(* PLC project LorochCxPlc_1, Beckhoff Automation GmbH TwinCAT PLC Control 3.5.13.20 *)
(* stored: creationDateTime 2021-05-25T13:03:07.2332886, modificationDateTime 2021-05-25T13:03:07.2402695 *)

FUNCTION_BLOCK FB_SFC_CHIPBREAKER_AUTO
(*---------------------------------------------------------------------------------------------------------------------------------------------------------------------------

			Date	I	version	I	remarks
					I			I
					I			I
					I			I
----------------------------------------------------------------------------------------------------------------------------------------------------------------------------*)
VAR_INPUT
				(*Positionierung Manuelle*)
				YDistanceToTouchPos					:	LREAL;
				ManPosActive							:	BOOL;
				XMoveManual							:	BOOL;
				SimpleTouch								:	BOOL;			(*Only 1 Touch*)
				KeyNextStep								:	BOOL;
				YrefPos									:	LREAL;			(*Reference Position  of Y-Axis)*)
				DoubleTouch								:	 BOOL;
				WorkingAngle							:	LREAL;
				Reset									:	 BOOL;
				PauseSwitchActive						:	 BOOL;
				MachineStateSafetyStateActive				:	 BOOL;
				MachineStateSharpenerDoorIsClosed		:        	BOOL;
				Start										:	 BOOL;
				AutomaticMode							:	 BOOL;
				ActualSawBlade							:	ST_SawBlade;
				ActualGrindingWheel						:	ST_GrindingWheel;
				ActualJob								:	ST_Job;
				AStartPos								:	 LREAL;				(*Rear Pos*)
				ChamferSideString						:	 STRING;
				ToothPitch								:	 LREAL;
				GrindingDirCW							:	 BOOL;
				DeltaMax								:	LREAL;
				TeethNumber								:	 INT;
				Stepper									:	 BOOL;							(*Using Servo Motor*)
				CbaPneumatic							:	BOOL;
				Zx										:	LREAL;							(*Z_Axis Corrector*)
				(*stepper-servo*)
				MarginRearValue							:	LREAL;							(*this value: Randabstand rear side to be set by the user*)
				MarginFrontValue							:	LREAL;							(*this value: Randabstand front side to be set by the user*)
				CbaMotionType							:	E_MotionType;
END_VAR
VAR_OUTPUT
				ActualStep								:	 INT;
				ErrorID									:	 DINT;
				ErrorOut									:	 BOOL;
				Paused									: 	BOOL;
				PauseRequest							:	 BOOL;
				PauseAvailable							:	 BOOL;
				CammingActive							:	 BOOL;
				ActualRevolutions							:     	UINT;
				ZStartposBuffered							:	 LREAL;
				ActualInfeed								:	LREAL;							(* actual infeed *)
				PartialInfeed								:	LREAL;
				ToothCount								:	INT;
				ZaxisCbaLimit							:	BOOL;
				CBAutoNotPossibleWithTooLargeSbDiameter	:	BOOL;
				WarningAaxisIsSlow						:	BOOL;
				CbaSpindleLowSpeedOutput				:	BOOL;

END_VAR

VAR_IN_OUT
				Done									:	BOOL;
				TouchPositionZAxis						:	LREAL;
				ChipBreakerAutoVeloTemp					:	LREAL;
				ChipBreakerManVeloOverrideFactor			:	LREAL;
END_VAR

VAR
				(*Manual Positionning*)
				RTrigConfirmTouchposZ					:	 R_TRIG;
				RTrigConfirmTouchposX					:	 R_TRIG;
				TON_Wait								:	 TON;
				DeltaXChamfering							:	 LREAL;
				ActualTeeth								:	 INT;
				SfcChipBreakerAuto						:	 FB_SUBFUNC_SEQ_CONTROL;	(* FB sfc *)
				XAxisStartPosition 							:	 LREAL;
				ZAxisStartPosition							:	 LREAL;
				ChipBreakerRear							:	 BOOL;
				StepNew									:	 INT;
				StepAction								:	 BOOL;
				StepActionImPulse						:	 BOOL;
				PauseStep								:	 INT;
				WorkingStepNo							:	 INT;
				AxisState								:	 E_StateMachineAxis;				(* check state of axis *)
				SBCircumference							:	 LREAL;
				ChipBreakerXAxisVelo						:	 LREAL;
				ChipBreakerAutoXAxisMaxVelo				: 	 LREAL;
				YAxisStartPosition							:	 LREAL;
				DegPerTeeth								:	 LREAL;
				XAxisTouchposRadio						:	 LREAL;
				TouchCorrection							:	 LREAL;
				FBCalcXOffset							:	 LREAL;
				XOffset									:	 LREAL;
				ZOffset									:	 LREAL;
				VarioCtr									:	 INT;
				VarioCtrEnd								:	 INT;
				XAxisEndPos								:	 LREAL;
				ZTouchPos								:	 LREAL;
				NumberTouch							:	 INT ;
				Delta									:         LREAL;			(*ABS(TP1-TP2)*)
				NominalTeeth							:	 LREAL;
				PauseRequested							:	 BOOL;
				PartialInfeedChangedDownfeed				:	 BOOL;
				ZAxisPausePos							:	 LREAL;
				InfeedZAxisMM							:	 LREAL;
				TouchPositionsZPlausi						:	 ARRAY[0..2] OF LREAL;
				TouchPositionsPlausibilityOK				:	 BOOL;
				TouchPositionsPlausibilityError				:	 BOOL;
				ChipBreakerFront							:	 BOOL;
				XaxisEndPOsFront						:	 LREAL;			(*X-Axis End Position After The Sharpening *)
				DeltaX									:	 LREAL;
				DeltaZ									:	 LREAL;
				YendPos								:	 LREAL;			(*End Position Y-Axis after Grinding*)
				ZAxisUpfeedMM							:	 LREAL;
				ZAxisUpfeedPosition						:	 LREAL;
				WorkingAngleRAD						:	 LREAL;
				RSS									:	 LREAL;
				BSS										:	 LREAL	;
				ChipBreakerFr							:	 BOOL	:=	TRUE;
				ChipBreakerRe							:	 BOOL	:=	FALSE ;
				NumberRevolution						:	 INT:=0	     ;
				ActualGrindingWheelThickness				:	 LREAL;
				(*Enumeration added*)
				RTrigNextStep							:	R_TRIG;
				ContinousMode							:	 BOOL;
				NextStepPulse							:	BOOL;
				XPosition								:	LREAL;
				ZPosition								:	LREAL;
				TON_Rear								:	TON;							(*Delay before the start of the Rear Side*)
				TONWaitSafetyStatePause					:	TON;
				FTRIG_STOP							:	F_TRIG;
				DeltaX_DEG								:	LREAL;
				XoffsetInGrad								:	LREAL;
				TonWaitClamping							:	TON;
				Test										:	BOOL;
				StopChipBreaker							:	BOOL;
				StartButton								:	R_TRIG;
				Stop_Manual_Pos							:	F_TRIG;
				DSSDiff									:	LREAL;
				ZPosAfterSharpening						:	LREAL;
				(*Software Limit S*)
				ZAxisLimitPos							:	BOOL;
				R_TRIG_ZlimitPos							:	R_TRIG;
				CbaLimit									:	BOOL;
				WaitAfterPause							:	TON;
				(*Vario*)
				VarioToothPitch							:	ARRAY[0..11] OF LREAL;
				VarioCtrFront1							:	INT;
				VarioCtrFront2							:	INT;
				VarioCtrRear1							:	INT;
				VarioCtrRear2							:	INT;
				GearPlayXAxis							:	LREAL;
				DifferenceMaxMinCBAGWDiameter			:	LREAL;
				(*Display Warning*)
				UIEventCBAProtection						:	FB_SUBFUNC_MESSAGE;
				ChipBreakerAutoGWwidth					:	LREAL;
				AaxisReferenceValue						:	LREAL;    (*the initial distance in MM when the axis is in home position*)
				AFront80									:	LREAL;	(*80% of the A-Axis front destination*)
				ARear80									:	LREAL;	(*80 % of the A -Axis Rear position *)
				AaxisRef80								:	LREAL;	(**)
				ARearPos								:	LREAL;
				AFrontPos								:	 LREAL;
				TonMonitoringAaxis						:	TON;
				StartMonitoringAaxis						:	BOOL;
				WarningAaxis								:	BOOL;
				RtrigAaxisIsTooSlow						:	R_TRIG;
				RtrigSpindleLowSpeedError				:	R_TRIG;
				CbaSpindleLowSpeed						:	BOOL;
				TriesNumber								:	INT;  (*Number of tries to find out the Reference position of A-axis*)
				AaxisRefPosTemp						:	LREAL;
				AaxisActPosition							:	LREAL;
				StartMovingStepByStepRear				:	BOOL; (**)
				StartMovingStepByStepFront				:	BOOL;
				ZTouchPosFirstTouchPos					:	LREAL;
				AaxisStepPositionIsReached				:	BOOL;
				WaitForAaxis								:	TON;
				StartWaitAaxis							:	BOOL;
				ZaxisFirstTouchPos						:	LREAL;
				ZNoTouch								:	LREAL;
				LastZPos								:	LREAL;
				LimitZaxis								:	LREAL;
				Zcomp									:	LREAL;
				StepperResults							:	FB_StepperResults;
				FileNameExtension						:	T_MaxString;
				StartWriting								:	BOOL;
				FileName								:	STRING;
				stTimeStruct								: 	TIMESTRUCT;
				stTimeStartM								: 	TIMESTRUCT;
				stTimeEndM								: 	TIMESTRUCT;
				ZposForCsv								:	LREAL;
				DurationAaxisMotion						:	TIME;
				StartTimeCounting							:	BOOL;
				TonCounting								:	TP;
				fbGetTime								: 	NT_GetTime;
				FirstEdgePos								:	LREAL;
				TestZ									:	BOOL;
				SecondEdge								:	LREAL;
				StepMotorNeededTimeToMove				:	TIME;
				StepMotorDestination						:	LREAL;
				AaxisTolerenceFast						:	LREAL;
				AaxisTolerenceSlow						:	LREAL;
				RTrigMonitoringCrash						:	R_TRIG;
				MonitoringTouchBack						:	LREAL;
				MonitoringTouchFront						:	LREAL;
				OperatingDirection						:	ST_OperatingDirection;
				TestCW									:	BOOL;
				TestCCW								:	BOOL;
				CalculatedXPosition,DiffXactposXcalcPos		:	LREAL;
				NumberOfTeethToAddReal					:	LREAL;
				NumberOfTeethToAdd						:	INT;
				rValueToAdd								:	LREAL;
				NombreOfRevolution						:	INT;
				GearPlayXAxisSharpChamfer				:	LREAL;
				(* Compensation *)
				NoOfActTeethCompensation				:	INT;
				XAxisNextPosition							:	LREAL;
				TestArray								:	ARRAY[0..5] OF BOOL;
END_VAR

            
	(* ---------------------------------------------------------------------------- SFC CHIPBREAKER AUTO -------------------------------------------------------------------------- *)

	(* call sfc functionblock *)
	SfcChipBreakerAuto(
						StepNew			:=	StepNew ,
						Reset			:=	Reset ,
						Step			=>	ActualStep ,
						StepAction		=>	StepAction ,
						StepActionImPulse=>	StepActionImPulse			 );


	TestZ			:=	TRUE;

	ContinousMode      := 	TRUE; 	   ;	(*TRUE; ;*)


	(*Reset the Sfc Variables*)
	IF	Reset
		THEN
			CbaSpindleLowSpeed														:=	FALSE;
			CbaSpindleLowSpeedOutput												:=	FALSE;
			StepNew																	:= 	0;
			Done																	:=	FALSE;
			ErrorOut																	:=	FALSE;
			ErrorID																	:=	0;
			StopChipBreaker															:=	FALSE;
			ZaxisCbaLimit															:=	FALSE;
			CBAutoNotPossibleWithTooLargeSbDiameter									:=	FALSE;
			MachineCtrl.Peripheral.ChipBreaker.Auto.DustFan.CmdOn						:=	FALSE;
			MachineCtrl.Peripheral.ChipBreaker.Auto.LowSpeedMonitoring.IsDeactivated		:=	FALSE;
			WarningAaxis																:=	FALSE;
			WarningAaxisIsSlow														:=	FALSE;
			MachineCtrl.ProcessControl.Warning.No										:=	0;
			StartTimeCounting															:=	FALSE;
			RTrigMonitoringCrash(CLK:=FALSE);
			MachineCtrl.State.ChipBreaker.Auto.GrindingWheelIsReady						:=	FALSE;
	END_IF;

			ChipBreakerAutoGWwidth			:=		UI.MachineSpecification.PeripheralOptional.ChipBreaker.GrindingWheel.Width.Nominal;

			AaxisTolerenceSlow				:=		0.01;
			AaxisTolerenceFast				:=		0.03;

			(*Edge distance  from ui*)


			MarginRearValue					:= 	UI.Order.Job[UI.State.ActualValues.ActualJobNumber.Maximal -1].EdgeDistance.EdgeDistanceRear;
			MarginFrontValue					:= 	UI.Order.Job[UI.State.ActualValues.ActualJobNumber.Maximal -1].EdgeDistance.EdgeDistanceFront;;


	(*###############################################A-Stepper Monitoring###############################################*)
			IF	(AxisCtrl[AxisNo.AAxis].Command.NominalValue.VeloJog <> 0)
				THEN
					IF	(StepNew <> 5030) AND
						(StepNew <> 5090)AND
						(StepNew <> 5100)
						THEN
							StepMotorNeededTimeToMove		:=
																		LREAL_TO_TIME(( ABS( AaxisActPosition -
																						StepMotorDestination ) /
																						AxisCtrl[AxisNo.AAxis].Command.NominalValue.VeloJog) );
																	;
						ELSE
							StepMotorNeededTimeToMove		:=	TIME#0.1s;
					END_IF;
				ELSE
					StepMotorNeededTimeToMove		:=	TIME#0.1s;
			END_IF;

			TonMonitoringAaxis(IN:= StartMonitoringAaxis , PT:= (StepMotorNeededTimeToMove*1000)+TIME#4s , Q=> , ET=> );


			RtrigAaxisIsTooSlow(CLK	:=	TonMonitoringAaxis.Q  , Q=> );

	(*Generate an error if the A-Axis is slow or not moving*)

	IF	RtrigAaxisIsTooSlow.Q
		THEN
			StepNew					:=	31000;
			TonMonitoringAaxis(  IN	:=	FALSE);
			RtrigAaxisIsTooSlow(CLK	:=	FALSE);
			StartMonitoringAaxis		:=	FALSE;
			WarningAaxis				:=	TRUE;
	END_IF;

	(*############################################A-Stepper Monitoring End##############################################*)

			StartButton(CLK:= MachineCtrl.Peripheral.ExternalControl.StartSwitch , Q=> );

		(*Manual Positionning*)

			ManPosActive	:=	MachineCtrl.Peripheral.ChipBreaker.Auto.PositionningMode.ManualPositionningIsActive;


		(*---------Software Limit--------------*)

			R_TRIG_ZlimitPos	(CLK :=	ZAxisLimitPos , Q=> );


		(*Controlling Z-Axis Limit Position*)
		IF	R_TRIG_ZlimitPos.Q
			THEN
				StepNew		:=	31000;
				CbaLimit		:=	TRUE;
		END_IF;

		(*Stop Button *)

		Stop_Manual_Pos(CLK:=	 (NOT PauseSwitchActive) , Q=> );

		FTRIG_STOP(CLK	:=	 (NOT PauseSwitchActive) ,
								   Q		=>		 );

		(*Z-Axis Confirm Touch Pos*)
		RTrigConfirmTouchposZ(CLK	:=	MachineCtrl.Peripheral.ExternalControl.ConfirmTouchpos	 , Q=> );

		(*X-Axis Confirm Touch Pos*)
		RTrigConfirmTouchposX(CLK	:= 	MachineCtrl.Peripheral.ExternalControl.ConfirmTouchpos, 	Q=> );


		IF	(StepNew	= 9815)
			THEN
				StartTimeCounting		:=	TRUE;
		END_IF;


	TonCounting(IN:= StartTimeCounting , PT:=TIME#180s , Q=> , ET=> );

		IF	(StepNew	= 985)
			THEN
				StartTimeCounting		:=	FALSE;
				DurationAaxisMotion	:=	TonCounting.ET;
		END_IF;


		(* r_trig next step *)
		RTrigNextStep( CLK := KeyNextStep );
		(* no confirm *)
		(*ContinousMode := FALSE;*)

;
	(*------------------------------------------Pause Requeted---------------------------------------*)

IF	(SfcChipBreakerAuto.Step	<=	1350) AND
	(SfcChipBreakerAuto.Step	>=	1300) AND
		(* pause switch is pressed *)
	(NOT PauseSwitchActive)
		THEN
			PauseRequested		:=	TRUE;
	END_IF;


IF	(SfcChipBreakerAuto.Step	= 9815)
	THEN
		IF	FTRIG_STOP.Q
		THEN
			StepNew		:=	31000;				(*Stop Routine *)
	END_IF;
END_IF;


IF	((SfcChipBreakerAuto.Step	>	1350) OR
	(SfcChipBreakerAuto.Step	<	1300))  AND(*OR*)
	( (SfcChipBreakerAuto.Step	<	90) OR
	(SfcChipBreakerAuto.Step	>	170))
	THEN
		IF	FTRIG_STOP.Q
			THEN
				StepNew		:=	31000;				(*Stop Routine *)
		END_IF;
END_IF;


IF	(SfcChipBreakerAuto.Step >=90)  AND
	(SfcChipBreakerAuto.Step <=170) AND
	Stop_Manual_Pos.Q
	THEN

				StepNew		:=	31600;				(*Direct Stop*)
END_IF;

	(*---------------------------------------ERROR------------------------------------------*)
	(*Error*)
	IF	(ChipBreakerFr AND
		ChipBreakerRe) OR
		( CbaPneumatic AND
		 Stepper)
		THEN
			StepNew		:=	25000;		(*Error*)
	END_IF;

	(* --------------------------------------sfc Reset----------------------------------------- *)

	IF	Reset
		THEN
			StepNew																	:= 	0;
			Done																	:=	FALSE;
			ErrorOut																	:=	FALSE;
			ErrorID																	:=	0;
			StopChipBreaker															:=	FALSE;
			ZaxisCbaLimit															:=	FALSE;
			CBAutoNotPossibleWithTooLargeSbDiameter									:=	FALSE;
			MachineCtrl.Peripheral.ChipBreaker.Auto.DustFan.CmdOn						:=	FALSE;
			MachineCtrl.Peripheral.ChipBreaker.Auto.LowSpeedMonitoring.IsDeactivated		:=	FALSE;
			WarningAaxis																:=	FALSE;
			AaxisStepPositionIsReached												:=	FALSE;
			StartWaitAaxis															:=	FALSE;
			ZNoTouch																:=	0;
			 MachineCtrl.Peripheral.ChipBreaker.Auto.LowSpeedMonitoring.ErrorOccured 		:=	FALSE;
			RTrigMonitoringCrash(CLK:=FALSE);
			MachineCtrl.State.ChipBreaker.Auto.GrindingWheelIsReady						:=	FALSE;
	END_IF;






	(*Test low speed warning and instead error*)

	RtrigSpindleLowSpeedError(CLK:= MachineCtrl.Peripheral.ChipBreaker.Auto.LowSpeedMonitoring.ErrorOccured , Q=> );

	IF	RtrigSpindleLowSpeedError.Q
		THEN
			 StepNew			:=	31000;
			CbaSpindleLowSpeed	:=	 TRUE;
	END_IF;



	ZAxisLimitPos		:=	(Axis[AxisNo.ZAxis].NcToPlc.ActPos <=  (UI.Order.SawBladeHolder.SawBladeLimitation[SBHChipBreakerAutoProtectionIndex].SawBladeDiameter.Minimal)) AND
							(StepNew >=85);

	(*---------------------------------------- pause------------------------------------------- *)

	IF	(SfcChipBreakerAuto.Step	<=	1350) AND
		(SfcChipBreakerAuto.Step	>=	1300)
		THEN
		IF	PauseAvailable AND
			(* pause switch is pressed *)
			(NOT PauseSwitchActive)
			THEN
				PauseRequested			:=	TRUE;
		END_IF;
	END_IF;



	CASE	SfcChipBreakerAuto.Step	OF

		(*------------------------------------------------------------------------ init Step - Reset all------------------------------------------------------------------------  *)
	0	:		(* action: predefine values *)
					CBAutoNotPossibleWithTooLargeSbDiameter							:=	FALSE;
					IF	StepActionImPulse
						THEN
							(* set axis state for check *)
								AxisState	:=	STATE_DISABLED;

							(* Reset x-axis *)
								AxisCtrl[AxisNo.XAxis].Command.OperationMode.CmdPowerOn				:=	FALSE;
								AxisCtrl[AxisNo.XAxis].Command.OperationMode.CmdMoveAbsolut			:=	FALSE;
								AxisCtrl[AxisNo.XAxis].Command.OperationMode.CmdCamming				:=	FALSE;

							(* Reset Z-axis *)
								AxisCtrl[AxisNo.ZAxis].Command.OperationMode.CmdPowerOn				:=	FALSE;
								AxisCtrl[AxisNo.ZAxis].Command.OperationMode.CmdMoveAbsolut			:=	FALSE;
								AxisCtrl[AxisNo.ZAxis].Command.OperationMode.CmdCamming				:=	FALSE;
							(*Reset A-Axis*)
								AxisCtrl[AxisNo.AAxis].Command.OperationMode.CmdPowerOn				:=	FALSE;
								AxisCtrl[AxisNo.AAxis].Command.OperationMode.CmdMoveAbsolut			:=	FALSE;
								AxisCtrl[AxisNo.AAxis].Command.OperationMode.CmdCamming				:=	FALSE;
								AxisCtrl[AxisNo.AAxis].Command.OperationMode.CmdJog					:=	FALSE;

								MachineCtrl.Peripheral.ChipBreaker.Auto.DustFan.CmdOn					:=	FALSE;
								CBAutoNotPossibleWithTooLargeSbDiameter								:=	FALSE;
								MachineCtrl.State.ChipBreaker.Auto.PauseIsActive							:=	FALSE;
								MachineCtrl.Peripheral.ExternalControl.StatusLedOnTouch1					:=	FALSE;
								MachineCtrl.Peripheral.ExternalControl.StatusLedOnTouch2					:=	FALSE;

								MachineCtrl.Peripheral.ChipBreaker.Auto.LowSpeedMonitoring.IsDeactivated	:=	FALSE;
								 MachineCtrl.Peripheral.ChipBreaker.Auto.LowSpeedMonitoring.ErrorOccured 	:=	FALSE;

								Done						:=	FALSE;
								ErrorOut						:=	FALSE;
								ErrorID						:=	0;
								ActualTeeth					:=	0;
								Paused						:=	FALSE;
								PauseStep					:=	0;
								PauseAvailable				:=	FALSE;
								PauseRequest				:=	FALSE;
								PauseRequested				:=	FALSE;
								WorkingStepNo				:=	1;
								CammingActive				:=	FALSE;
								NumberTouch				:=	0;
								Delta						:=	0;
								NumberRevolution			:=	0;
								SimpleTouch					:=	FALSE;				(*OnlyOne Touch*)
								DoubleTouch					:=	FALSE;				(*We Requie 2 Touchs*)
								ErrorOut						:=	FALSE;
								NumberTouch				:=	0;
								ActualRevolutions				:=	0;
								StopChipBreaker				:=	FALSE;
								KeyNextStep					:=	FALSE;
								(*Positionning Type*)
								ManPosActive				:=	FALSE;
								(* status led touching *)
								CbaSpindleLowSpeed			:=	FALSE;
								CbaSpindleLowSpeedOutput	:=	FALSE;
								StopChipBreaker				:=	FALSE;
								CbaLimit						:=	FALSE;
								ZaxisCbaLimit				:=	FALSE;
								WarningAaxis					:=	FALSE;
								WarningAaxisIsSlow			:=	FALSE;
								StartMonitoringAaxis			:=	FALSE;
								StartMovingStepByStepRear	:=	FALSE;
								StartMovingStepByStepFront	:=	FALSE;
								TriesNumber					:=	0;
								AaxisStepPositionIsReached	:=	FALSE;
								StartWaitAaxis				:=	FALSE;
								ZNoTouch					:=	0;
								ZposForCsv					:=	0;
								StartWriting					:=	FALSE;
								RTrigMonitoringCrash(CLK:=FALSE);
								TestCW						:=	FALSE;
								TestCCW					:=	FALSE;
					END_IF;

					(* transition *)
					IF	StepAction AND
						(NOT StepActionImPulse) AND
						(* stop switch not pressed *)
							PauseSwitchActive
						THEN
							StepNew	:= 10;									(* -> wait for Start *)
					END_IF;
		(*-------------------------------------------------------------  wait for Start----------------------------------------------------------------- *)
	10	:
					(* transition:  *)
					IF	StepAction AND
						(NOT StepActionImPulse) AND
						(* recut/resharp only in automatic mode *)
							AutomaticMode AND
						(* Start sfc from external *)
							Start AND
						(* machine door is closed *)
							MachineStateSharpenerDoorIsClosed AND
						(* safe state are disabled *)
							(NOT MachineStateSafetyStateActive) AND
						 (* stop switch not pressed *)
							(PauseSwitchActive)
						THEN
							StepNew									:= 	20;									(* -> Enable X-axis ,Z-axis and A -Axis*)
							ChipBreakerFr							:=	TRUE;
							ChipBreakerRe							:=	FALSE;
							StopChipBreaker							:=	FALSE;
							KeyNextStep								:=	FALSE;
							ErrorOut									:=	FALSE;
							ZaxisCbaLimit							:=	FALSE;
							CBAutoNotPossibleWithTooLargeSbDiameter	:=	FALSE;
							AaxisRefPosTemp						:=	UI.MachineSpecification.PeripheralOptional.ChipBreaker.Notch.SBEdgeOffset;			(*Reference Value of the A-Axis*)
							AaxisReferenceValue						:=	AaxisRefPosTemp;
							AaxisStepPositionIsReached				:=	FALSE;
							StartWaitAaxis							:=	FALSE;
							ZNoTouch								:=	0;
							StartWriting								:=	FALSE;
							 MachineCtrl.Peripheral.ChipBreaker.Auto.LowSpeedMonitoring.ErrorOccured 	:=	FALSE;
							MachineCtrl.State.ChipBreaker.Auto.GrindingWheelIsReady					:=	FALSE;
					END_IF;

		(*------------------------------------------------------------Wait For User Interaction--------------------------------------------------------------*)
	20:			IF	StepActionImpulse
					THEN
						NextStepPulse		:=	TRUE;
					END_IF;

				IF	StepAction AND
					( RTrigNextStep.Q OR
					ContinousMode )
					THEN
						StepNew				:= 	22;
						NextStepPulse		:=	FALSE;
						ErrorOut				:=	FALSE;
				END_IF;

		(*---------------------------------------------------------------- action: Enable x +z+a Axis-----------------------------------------------------------*)
	22	:		(*Action*)
					ErrorOut					:=	FALSE;
					IF	StepActionImPulse
						THEN
							(* set axis state for check *)
								AxisState	:=	STATE_WAIT_NEWOPERATION;
							(* x-axis - Enable *)
								AxisCtrl[AxisNo.XAxis].Command.OperationMode.CmdPowerOn			:=	TRUE;
								AxisCtrl[AxisNo.XAxis].Command.OperationMode.CmdMoveAbsolut		:=	FALSE;
								AxisCtrl[AxisNo.XAxis].Command.OperationMode.CmdCamming			:=	FALSE;
								AxisCtrl[AxisNo.XAxis].Command.ExternalControl.override				:=	100;
							(* Z-axis - Enable *)
								AxisCtrl[AxisNo.ZAxis].Command.OperationMode.CmdPowerOn			:=	TRUE;
								AxisCtrl[AxisNo.ZAxis].Command.OperationMode.CmdMoveAbsolut		:=	FALSE;
								AxisCtrl[AxisNo.ZAxis].Command.OperationMode.CmdCamming			:=	FALSE;
								AxisCtrl[AxisNo.ZAxis].Command.ExternalControl.override				:=	100;
							(* Axis Is Used--> Axis Enable*)
								IF	Stepper
									THEN
							(*A-Axis- Enable*)
								AxisCtrl[AxisNo.AAxis].Command.OperationMode.CmdPowerOn			:=	TRUE;
								AxisCtrl[AxisNo.AAxis].Command.OperationMode.CmdMoveAbsolut		:=	FALSE;
								AxisCtrl[AxisNo.AAxis].Command.OperationMode.CmdCamming			:=	FALSE;
								AxisCtrl[AxisNo.AAxis].Command.ExternalControl.override				:=	100;
								END_IF;
						END_IF;

					(* transition: axis are Enabled? *)
					IF	StepAction AND
						(NOT StepActionImPulse)
						THEN
							IF	Stepper
								THEN
						(* recut/resharp only in automatic mode *)
								IF	AutomaticMode AND
								(* status x-axis *)
									(NOT Axis[AxisNo.XAxis].Status.Disabled) AND
									Axis[AxisNo.XAxis].Status.StandStill AND
									( AxisCtrl[AxisNo.XAxis].feedback.state.ActualFbState = AxisState ) AND
								(* status Z-axis *)
									(NOT Axis[AxisNo.ZAxis].Status.Disabled) AND
									Axis[AxisNo.ZAxis].Status.StandStill AND
									( AxisCtrl[AxisNo.ZAxis].feedback.state.ActualFbState = AxisState ) AND
								(*Status A-Axis*)
									(NOT Axis[AxisNo.AAxis].Status.Disabled) AND
									Axis[AxisNo.AAxis].Status.StandStill AND
									( AxisCtrl[AxisNo.AAxis].feedback.state.ActualFbState = AxisState )AND
								(* stop switch not pressed *)
									(PauseSwitchActive)
									THEN
									StepNew	:= 	25;
								END_IF;
							ELSIF	CbaPneumatic
									THEN
										IF	AutomaticMode AND
											(* status x-axis *)
												(NOT Axis[AxisNo.XAxis].Status.Disabled) AND
												Axis[AxisNo.XAxis].Status.StandStill AND
												( AxisCtrl[AxisNo.XAxis].feedback.state.ActualFbState = AxisState ) AND
											(* status Z-axis *)
												(NOT Axis[AxisNo.ZAxis].Status.Disabled) AND
												Axis[AxisNo.ZAxis].Status.StandStill AND
												( AxisCtrl[AxisNo.ZAxis].feedback.state.ActualFbState = AxisState ) AND
											(* stop switch not pressed *)
												(PauseSwitchActive)
												THEN
													StepNew		:=	25;	(*Wait for user Interaction*)
										END_IF;
							END_IF;
					END_IF;

(* ---------------------------------- wait for user interaction  ------------------------------------------- *)
	25:			IF	StepActionImpulse
					THEN
						NextStepPulse	:=	TRUE;
				END_IF;

				IF	StepAction AND
					( RTrigNextStep.Q OR
					ContinousMode )
					THEN
						StepNew			:= 	26;(*27*)
						ChipBreakerFr	:=	TRUE;
						ChipBreakerRe	:=	FALSE;
						NextStepPulse	:=	FALSE;
						ActualTeeth		:=	0;
						NumberTouch	:=	0;
						ErrorOut			:=	FALSE;
						StopChipBreaker	:=	FALSE;
						KeyNextStep		:=	FALSE;
				END_IF;

	(*--------------------------------------------Check Coolant Pump----------------------------------------------------------*)

	26:			(*Action*)
				IF	StepActionImPulse AND
					MachineCtrl.state.CoolantPump.unit.IsActive
					THEN
						MachineCtrl.Peripheral.CoolantPump.auto.CmdOn	:=	FALSE;
						MachineCtrl.Peripheral.CoolantPump.auto.CmdOff	:=	TRUE;
				END_IF;
		
				(* transition: coolant pump is disabled? *)
				IF	StepAction AND
					( NOT StepActionImPulse )
					THEN
						StepNew		:=	27;
				END_IF;

	(* ----------------------------------------------- move y-axis to position 0 : Ref--------------------------------------- *)
	27	:	(* action: move y-axis to position 0 *)
				IF	StepActionImPulse
					THEN
						(* y-axis *)
							AxisState														:=	STATE_WAIT_NEWOPERATION;
							AxisCtrl[AxisNo.YAxis].Command.OperationMode.CmdPowerOn			:=	TRUE;
							AxisCtrl[AxisNo.YAxis].Command.OperationMode.CmdMoveAbsolut		:=	TRUE;
							AxisCtrl[AxisNo.YAxis].Command.NominalValue.VeloMoveAbsolut		:=	30;			(*  mm / second *)
							AxisCtrl[AxisNo.YAxis].Command.NominalValue.PositionMoveAbsolut		:=	0;
							AxisCtrl[AxisNo.YAxis].Command.ExternalControl.Override				:=	100;
				END_IF;

				TON_Wait(IN:=		StepAction	AND
									(NOT StepActionImPulse) AND
									(* status y-axis *)
									Axis[AxisNo.YAxis].Status.StandStill AND
									Axis[AxisNo.YAxis].Status.InTargetPosition AND
									( AxisCtrl[AxisNo.YAxis].feedback.state.ActualFbState = AxisState ) AND
									( NOT AxisCtrl[AxisNo.YAxis].Command.OperationMode.CmdMoveAbsolut )		 ,
									 PT:=	TIME#3S
									 , Q=> , ET=> );
				(*Transition*)
				IF	StepAction	AND
					(NOT StepActionImPulse) AND
					(* status y-axis *)
					Axis[AxisNo.YAxis].Status.InTargetPosition AND
					( AxisCtrl[AxisNo.YAxis].feedback.state.ActualFbState = AxisState ) AND
					( NOT AxisCtrl[AxisNo.YAxis].Command.OperationMode.CmdMoveAbsolut )
					THEN
					StepNew		:=	28;
					AxisCtrl[AxisNo.YAxis].Command.OperationMode.CmdPowerOn			:=	FALSE;
					AxisCtrl[AxisNo.YAxis].Command.OperationMode.CmdMoveAbsolut		:=	FALSE;
				END_IF;
	(*-------------------------------------------------------Check Grinding Head Position---------------------------------------------------*)

	28:			(* action: grinding head to middle position *)
					IF	StepActionImPulse AND
						(* Grinding Head Not in Middle *)
						 ( NOT MachineCtrl.state.GrindingHead.Unit.IsInMiddlePosition )
						THEN
							MachineCtrl.Peripheral.GrindingHead.unit.auto.CmdMiddlePosition	:=	TRUE;
							MachineCtrl.Peripheral.GrindingHead.KeyLED.CmdMiddlePosition	:=	TRUE;
					END_IF;

					(* transition *)
					IF	StepAction AND
						(NOT StepActionImPulse) AND
						(* status grinding head *)
						( MachineCtrl.state.GrindingHead.Unit.IsInMiddlePosition )AND
						( NOT MachineCtrl.Peripheral.GrindingHead.unit.auto.CmdMiddlePosition )
						THEN
							StepNew	:= 29;				(*Check The Grinding Wheel Status*)
					END_IF;
	(*--------------------------------------------------------------Check The Grinding Wheel-----------------------------------------------------*)
	29:				(*Action*)
					IF	StepActionImPulse AND
						MachineCtrl.State.GrindingWheel.Unit.IsActive
						THEN
							MachineCtrl.Peripheral.GrindingWheel.Unit.Auto.CmdOff	:=	TRUE;
							MachineCtrl.Peripheral.GrindingWheel.Unit.Auto.CmdOn	:=	FALSE;
					END_IF;
					(*Transition*)
					IF	StepAction  AND
						(NOT StepActionImPulse)
						THEN
							StepNew		:=	30;
					END_IF;
	(*------------------------------------------------------------Compensation If Necessary-------------------------------------------------------*)

		30:			(*Action*)
					IF	StepActionImPulse
						THEN
							IF	(MachineCtrl.ProcessTemp.ActualJobData.OperatingDirection.PreviousPrevious <>MachineCtrl.ProcessTemp.ActualJobData.OperatingDirection.Previous)
								THEN
									IF	 (MachineCtrl.ProcessTemp.ActualJobData.OperatingDirection.PreviousPrevious = 'ClockWise')
										THEN
											GearPlayXAxisSharpChamfer	:=	UI.MachineSpecification.PeripheralBasic.Axis.X.GearBacklash * -1;
										ELSE
											GearPlayXAxisSharpChamfer	:=	UI.MachineSpecification.PeripheralBasic.Axis.X.GearBacklash ;
									END_IF;
								ELSE
									GearPlayXAxisSharpChamfer			:=	0;
							END_IF;

						IF 	(MachineCtrl.ProcessTemp.ActualJobData.OperatingDirection.Previous  <>
																						MachineCtrl.ProcessTemp.ActualJobData.OperatingDirection.Actual)
							THEN
								GearPlayXAxis	:=	UI.MachineSpecification.PeripheralBasic.Axis.X.GearBacklash * -1;
							ELSE
								GearPlayXAxis	:=	0;
						END_IF;

						GearPlayXAxis		:=	GearPlayXAxis +
												GearPlayXAxisSharpChamfer		;
					END_IF;

					(*Transition*)
					IF	StepAction AND
						(NOT StepActionImPulse)
						THEN
							StepNew		:=	40;
					END_IF;
	(*################################POSITIONIERUNG MANUELLE################################*)

		40:			(*Action*)
					IF	StepAction AND
						(NOT StepActionImPulse)
						THEN
							IF	ManPosActive
								THEN
									StepNew		:=	50;				(*Manual Positionning *)
								ELSE
									StepNew		:=	42;				(*Auto Positionning*)
							END_IF;
					END_IF;

	(*--------------------------------------------------------------Calc X Pos Depending On Previous Job--------------------------------------------------------*)

		42:			IF	StepAction AND
						(NOT StepActionImPulse)
						THEN
							IF	(MachineCtrl.ProcessTemp.ActualJobData.OperatingMode.Previous= OperatingMode.Recutting) OR
								(MachineCtrl.ProcessTemp.ActualJobData.OperatingMode.Previous= OperatingMode.ReSharpening)
								THEN
										StepNew		:=	45 ;
									ELSIF	(MachineCtrl.ProcessTemp.ActualJobData.OperatingMode.Previous= OperatingMode.Chamfering) OR
											(MachineCtrl.ProcessTemp.ActualJobData.OperatingMode.Previous= OperatingMode.ChamferingAllTeeth)
										THEN
												StepNew		:=	48	;
							END_IF;
					END_IF;

	(*--------------------------------------------------------------Calculation of Touch Position x/z Axis-------------------------------------------------------------*)
		45:			(*Action*)
					IF	StepActionImPulse
						THEN
							Zx			:=	UI.MachineSpecification.PeripheralOptional.ChipBreaker.ZPosCorrectionResharpRecut*2;
							(*degree per tooth calc*)
							IF	MachineCtrl.ProcessTemp.ActualJobData.SpecialTooth.VarioTooth.IsActive
								THEN
									DegPerTeeth			:=	MachineCtrl.ProcessTemp.ActualJobData.SpecialTooth.VarioTooth.LengthDEG;
								ELSE
									DegPerTeeth			:=	360.0 / MachineCtrl.ProcessTemp.ActualOrderStackBuffer.ActualOrder.SawBlade.NumberOfTeeth;
							END_IF;

							(*UpfeedMM calc*)
							ZAxisUpfeedMM		:=	2*(MachineCtrl.ProcessTemp.ActualJobData.Job.Infeed.TotalInfeed + REAL_TO_LREAL( UI.MachineSpecification.PeripheralOptional.ChipBreaker.YOffSet));
							RSS				:=	MachineCtrl.ProcessTemp.ActualOrderStackBuffer.ActualOrder.GrindingWheel.Diameter / 2;
							DSSDiff				:=	200 - MachineCtrl.ProcessTemp.ActualOrderStackBuffer.ActualOrder.GrindingWheel.Diameter;
							WorkingAngle		:=	UI.MachineSpecification.Base.WorkingAngle;
							BSS					:=	ActualGrindingWheel.Layer.Thickness;
							WorkingAngleRAD 	:=	WorkingAngle / 180 * PI;
							YrefPos				:=	YDistanceToTouchPos  -
													UI.MachineSpecification.PeripheralBasic.Axis.Y.Position.HomingOffset;																			(*Ref Point Of Y Axis*)
							YendPos			:=	MachineCtrl.ProcessTemp.ActualJobData.OperatingMode.EndPosActOpMode.PosY_CBA;	(*Y End Position Buffered After The Resharpening Or Retoothing*)

							DeltaZ				:=	2*(YrefPos-YendPos)*COS(WorkingAngleRAD ) + Zx + DSSDiff*COS(WorkingAngleRAD )  ;									(*Z-Axis Corrector : Zx*)
							DeltaX				:=	SIN(WorkingAngleRAD )*(YendPos - YrefPos -100+RSS) + 0.5*(BSS-2);
							DeltaX_DEG			:=	( 360.0 / (ActualSawBlade.Diameter * PI) ) * DeltaX;										(*DeltaX MM2DEG*)

							XoffsetInGrad			:=	( 360.0 / (ActualSawBlade.Diameter * PI) ) * UI.MachineSpecification.PeripheralOptional.ChipBreaker.XOffSet;

							ZPosition			:=
													ActualSawBlade.Diameter +
													 DeltaZ ;

							XPosition			:=	Axis[AxisNo.XAxis].NcToPlc.ActPos + GearPlayXAxis  ;
					END_IF;
					(*Transition: Is The Calcualtion Finished?*)
					IF 	StepAction AND
						(NOT StepActionImPulse)
						THEN
							StepNew		:=	50;				(*MoveX & Z Axis To Definiert  Pos*)
					END_IF;

	(*------------------------------------------------------------------------CBA After Chamfering-----------------------------------------------------------------------------*)

		48:
					(*Action*)
					IF	StepActionImPulse
						THEN
							Zx						:=	UI.MachineSpecification.PeripheralOptional.ChipBreaker.ZPosCorrectionResharpRecut*2;
							(*degree per tooth calc*)
							(*DegPerTeeth				:=	(1/ UINT_TO_LREAL(UI.Order.SawBlade.NumberOfTeeth))  *360; *)

								(*degree per tooth calc*)
							IF	MachineCtrl.ProcessTemp.ActualJobData.SpecialTooth.VarioTooth.IsActive
								THEN
									DegPerTeeth			:=	MachineCtrl.ProcessTemp.ActualJobData.SpecialTooth.VarioTooth.LengthDEG;
								ELSE
									DegPerTeeth			:=	360.0 / MachineCtrl.ProcessTemp.ActualOrderStackBuffer.ActualOrder.SawBlade.NumberOfTeeth;
							END_IF;

							(*UpfeedMM calc*)
							ZAxisUpfeedMM			:=	2*(MachineCtrl.ProcessTemp.ActualJobData.Job.Infeed.TotalInfeed +  REAL_TO_LREAL (UI.MachineSpecification.PeripheralOptional.ChipBreaker.YOffSet));
							RSS					:=	MachineCtrl.ProcessTemp.ActualOrderStackBuffer.ActualOrder.GrindingWheel.Diameter / 2;
							DSSDiff					:=	200 - MachineCtrl.ProcessTemp.ActualOrderStackBuffer.ActualOrder.GrindingWheel.Diameter;
							WorkingAngle			:=	UI.MachineSpecification.Base.WorkingAngle;
							BSS						:=	ActualGrindingWheel.Layer.Thickness;
							WorkingAngleRAD 		:=	WorkingAngle / 180 * PI;
							YrefPos					:=	YDistanceToTouchPos  -
														UI.MachineSpecification.PeripheralBasic.Axis.Y.Position.HomingOffset;																		(*Ref Point Of Y Axis*)
							YendPos				:=	MachineCtrl.ProcessTemp.ActualJobData.OperatingMode.EndPosActOpMode.PosY_CBA;	(*Y End Position Buffered After The Resharpening Or Retoothing*)

							DeltaZ					:=	2*(YrefPos-YendPos)*COS(WorkingAngleRAD ) + Zx + DSSDiff*COS(WorkingAngleRAD ) ;									(*Z-Axis  Corrector : Zx*)
							DeltaX					:=	SIN(WorkingAngleRAD )*(YendPos - YrefPos -100+RSS) + 0.5*(BSS-2);
							DeltaX_DEG				:=	( 360.0 / (ActualSawBlade.Diameter * PI) ) * DeltaX;										(*DeltaX MM2DEG*)
							XoffsetInGrad				:=	( 360.0 / (ActualSawBlade.Diameter * PI) ) * UI.MachineSpecification.PeripheralOptional.ChipBreaker.XOffSet;
														(*IF Previous Job Is Chamfering*)


							ZPosition				:=
														ActualSawBlade.Diameter +
														 DeltaZ ;
						(*----------------------------------------------------------------------------------------------------------------------*)
						IF	MachineCtrl.ProcessTemp.ActualJobData.OperatingDirection.Previous = 'CounterClockWise'
								THEN
									(*Position if chamfer is ccw*)
									CalculatedXPosition			:=	MachineCtrl.ProcessTemp.ActualJobData.OperatingMode.EndPosActOpMode.PosX_CBA +
														     		  	(360 *  2 * MachineCtrl.Peripheral.ChipBreaker.Auto.Number_Rev_Chamf.Rev_Chamfering)   + GearPlayXAxis;
								ELSE
									(*Position if chamfer is cw*)
									CalculatedXPosition			:=	MachineCtrl.ProcessTemp.ActualJobData.OperatingMode.EndPosActOpMode.PosX_CBA -
														     			(360 *  2 * MachineCtrl.Peripheral.ChipBreaker.Auto.Number_Rev_Chamf.Rev_Chamfering)  - GearPlayXAxis;
							END_IF;

							(*Difference between Calculated Pos and Actual Pos after chamfering*)
							DiffXactposXcalcPos				:=	ABS (  CalculatedXPosition - MachineCtrl.ProcessTemp.ActualJobData.OperatingMode.EndPosActOpMode.PosX);
							(*convert this difference to number of teeth*)
							NumberOfTeethToAddReal			:= 	(DiffXactposXcalcPos / DegPerTeeth);

							IF  (	LMOD (DiffXactposXcalcPos , DegPerTeeth)   <> 0)
								THEN
									NumberOfTeethToAdd		:=	TRUNC_INT (NumberOfTeethToAddReal )+1;
								ELSE
									NumberOfTeethToAdd		:=	TRUNC_INT (NumberOfTeethToAddReal ) ;
							END_IF;

							(*Value for compensation *)
							rValueToAdd						:=	INT_TO_LREAL(NumberOfTeethToAdd) * DegPerTeeth;

							IF	(CalculatedXPosition <  MachineCtrl.ProcessTemp.ActualJobData.OperatingMode.EndPosActOpMode.PosX) (* Actpos X-Axis *)
								THEN
									XPosition			:=		CalculatedXPosition + rValueToAdd;
								ELSE
									XPosition			:=		CalculatedXPosition - rValueToAdd ;(* + DegPerTeeth - LMOD (DiffXactposXcalcPos , DegPerTeeth ) *) ;
									TestCW	:=	TRUE;

							END_IF;
					END_IF;
					(*Transition: Is The Calcualtion Finished?*)
					IF 	StepAction AND
						(NOT StepActionImPulse)
						THEN
							StepNew		:=	50;							(*MoveX & Z Axis To Definiert  Pos*)
					END_IF;

	(*-------------------------------------------------------Saw Blade Bracket To  Home Pos----------------------------------------------------------------------*)

		50:			(*Action*)
					IF	StepActionImPulse
						THEN
							IF	( NOT MachineCtrl.state.SawBladeBracket.InHomePosition)
								THEN
									MachineCtrl.Peripheral.SawBladeBracket.CmdWorkPos		:=	FALSE;
									MachineCtrl.Peripheral.SawBladeBracket.CmdHomePos	:=	TRUE;
							END_IF;
					END_IF;
					(*Transition is Saw Blade Bracket In Home Position ?*)

					IF StepAction AND
					     (NOT StepActionImPulse) AND
					     (NOT MachineCtrl.Peripheral.SawBladeBracket.CmdHomePos) AND
					      MachineCtrl.state.SawBladeBracket.InHomePosition
					THEN
							IF	ManPosActive
								THEN
									(* man positioning mode -> z-axis to handover pos *)
								(*	ZPosAfterSharpening	:=	UI.MachineSpecification.PeripheralBasic.Axis.Positions.HandOver;;*)
									StepNew				:=	75;
								ELSE
									(* auto positioning mode -> move z-axis down *)
									ZPosAfterSharpening	:=	Axis[AxisNo.ZAxis].NcToPlc.ActPos + 160  ;
									StepNew				:=	60;
							END_IF;

					END_IF;
	(*---------------------------------------------------------------Action Move  To Z Axis Handover Position----------------------------------------------------*)
	60	:			(*Action*)

					IF	 StepActionImPulse
						THEN
							(* Z-axis - move absolute *)
							AxisCtrl[AxisNo.ZAxis].Command.OperationMode.CmdPowerOn			:=	TRUE;
							AxisCtrl[AxisNo.ZAxis].Command.OperationMode.CmdJogHandwheel 		:=	FALSE;
							AxisCtrl[AxisNo.ZAxis].Command.OperationMode.CmdMoveAbsolut		:=	TRUE;
							AxisCtrl[AxisNo.ZAxis].Command.OperationMode.CmdCamming			:=	FALSE;
							AxisCtrl[AxisNo.ZAxis].Command.NominalValue.VeloMoveAbsolut		:=	100;
							IF	(ZPosAfterSharpening <=  UI.MachineSpecification.PeripheralBasic.Axis.Positions.Homing)  		(*To Avoid Going Deeper than Homing Position Z-Axis*)
								THEN
									AxisCtrl[AxisNo.ZAxis].Command.NominalValue.PositionMoveAbsolut		:=	ZPosAfterSharpening;
								ELSE
									CBAutoNotPossibleWithTooLargeSbDiameter		:=	TRUE;
							END_IF;
					END_IF;

					(*Transition : Is Z- Axis In Handover Pos?*)

					IF     	StepAction AND
					   	 (NOT StepActionImPulse) AND
						(Axis[AxisNo.ZAxis].NcToPlc.ActPos	>= ZPosAfterSharpening - 0.1) AND
						(Axis[AxisNo.ZAxis].NcToPlc.ActPos	<= ZPosAfterSharpening +0.1)
						THEN
							StepNew		:=	70;							(*ChipBreaker Swivel Unit To Work Pos*)
					END_IF;

		(*-----------------------------------------------------------------Wait For User Interaction-----------------------------------------------------------------*)

	70:			(*Action*)
				IF	StepActionImpulse
					THEN
						NextStepPulse	:=	TRUE;
				END_IF;

				IF	StepAction AND
					( RTrigNextStep.Q OR
					ContinousMode )
					THEN
						StepNew			:= 	80;
						NextStepPulse	:=	FALSE;
				END_IF;
                     (*  ----------------------------------------------------------------------------------------------------------------------------------------------------------------*)
	75:
				IF	StepActionImPulse
					THEN
					(* set axis state for check *)
						AxisState	:=	STATE_WAIT_NEWOPERATION;
					(* x-axis - Enable *)
						AxisCtrl[AxisNo.ZAxis].Command.OperationMode.CmdPowerOn			:=	TRUE;
						AxisCtrl[AxisNo.ZAxis].Command.OperationMode.CmdMoveAbsolut		:=	TRUE;
						AxisCtrl[AxisNo.ZAxis].Command.OperationMode.CmdCamming			:=	FALSE;
						AxisCtrl[AxisNo.ZAxis].Command.NominalValue.VeloMoveAbsolut		:=	20;
						AxisCtrl[AxisNo.ZAxis].Command.ExternalControl.override				:=	100;
						AxisCtrl[AxisNo.ZAxis].Command.NominalValue.PositionMoveAbsolut		:=	UI.MachineSpecification.PeripheralBasic.Axis.Positions.Homing;;
				END_IF;
				(*Transition : Is Z- Axis In Reference Pos?*)
				IF     	StepAction AND
				   	 (NOT StepActionImPulse) AND
					  (Axis[AxisNo.ZAxis].NcToPlc.ActPos >= UI.MachineSpecification.PeripheralBasic.Axis.Positions.Homing) AND
					  (NOT Axis[AxisNo.ZAxis].Status.Disabled)
					THEN
						StepNew		:=	80;
				END_IF;


		(*----------------------------------------------------Chip Breaker Swivel Unit  to Work Position------------------------------------------------#6*)
	80	:		(*Action *)
				IF 	StepActionImpulse AND
					(NOT MachineCtrl.State.ChipBreaker.Auto.SwivelUnit.InWorkPosition)
					THEN
						MachineCtrl.Peripheral.ChipBreaker.Auto.SwivelUnit.CmdHomePos	:=	FALSE;
						MachineCtrl.Peripheral.ChipBreaker.Auto.SwivelUnit.CmdWorkPos	:=	TRUE;
				END_IF;

				(*Transition : Is Chip Breaker In Work Position?*)

				IF 	StepAction AND
				   	 (NOT StepActionImPulse) AND
				     	MachineCtrl.State.ChipBreaker.Auto.SwivelUnit.InWorkPosition
					THEN
						StepNew		:=	82;		(*Release Clamping*)
				END_IF;
		(*--------------------------------------------------------------------Release Clamping-----------------------------------------------------------------------*)

	82:			(*Action*)
					IF	StepActionImPulse
						THEN
						MachineCtrl.Peripheral.ChipBreaker.Auto.Clamping.CmdClose	:=	FALSE;
						MachineCtrl.Peripheral.ChipBreaker.Auto.Clamping.CmdOpen	:=	TRUE;
					END_IF;

					(* transition:  *)
					IF	StepAction AND
						(NOT StepActionImPulse) AND
						MachineCtrl.State.ChipBreaker.Auto.Clamping.IsReleased
						THEN
							StepNew	:= 	85;			(*Select The Positionning Mode*)
					END_IF;

		(*----------------------------------------------------------------Wait For User Interaction---------------------------------------------------------------*)

	85:			IF	StepActionImpulse
					THEN
						NextStepPulse	:=	TRUE;
				END_IF;

				(*Transition*)
				IF	StepAction AND
					(NOT StepActionImPulse) AND
					( NOT MachineCtrl.state.GrindingWheel.unit.IsActive ) AND
					( NOT MachineCtrl.Peripheral.GrindingWheel.unit.auto.CmdOff ) AND
					( NOT MachineCtrl.Peripheral.CoolantPump.auto.CmdOff ) AND
					( NOT MachineCtrl.state.CoolantPump.unit.IsActive )
					THEN
						StepNew			:= 	86;		(* ManPosActive?*)
						NextStepPulse	:=	FALSE;
				END_IF;

		(*----------------------------------------------------------------------ManPosActive?--------------------------------------------------------------------*)

		(*Transition*)
	86:				IF	StepAction AND
						(NOT StepActionImPulse)
						THEN
							IF	ManPosActive
								THEN
									StepNew		:=	90;		(*Axe Deactivieren --> start of manual positionning*)
									ELSE
										StepNew		:=	875	(* Move Z & X Axis To Calculated  Positions*);
							END_IF;
					END_IF;

	(*####################################Manual Positionning#######################################*)


	(*--------------------------------------------------------------------deactivate axis Z&X---------------------------------------------------------------*)

	90:				(* action:   *)
				IF	StepActionImPulse
					THEN
						(* set axis state for check *)
							AxisState	:=	STATE_INIT;
						(* x-axis - disable *)
							AxisCtrl[AxisNo.XAxis].Command.OperationMode.CmdPowerOn			:=	FALSE;
							AxisCtrl[AxisNo.XAxis].Command.OperationMode.CmdMoveAbsolut		:=	FALSE;
							AxisCtrl[AxisNo.XAxis].Command.OperationMode.CmdCamming			:=	FALSE;
						(* z-axis - disable *)
							AxisCtrl[AxisNo.ZAxis].Command.OperationMode.CmdPowerOn			:=	FALSE;
							AxisCtrl[AxisNo.ZAxis].Command.OperationMode.CmdMoveAbsolut		:=	FALSE;
							AxisCtrl[AxisNo.ZAxis].Command.OperationMode.CmdCamming			:=	FALSE;
				END_IF;
				(* transition:  *)
				IF	StepAction AND
					(NOT StepActionImPulse) AND
					(* status x-axis *)
						Axis[AxisNo.XAxis].Status.Disabled AND
						( AxisCtrl[AxisNo.XAxis].feedback.state.ActualFbState = AxisState ) AND
					(* status z-axis *)
						Axis[AxisNo.ZAxis].Status.Disabled AND
						( AxisCtrl[AxisNo.ZAxis].feedback.state.ActualFbState = AxisState )
					THEN
						StepNew		:= 	95;			(*Reset X-Axis Act Position*)
					END_IF;

		(* ---------------------------------------------------------- reset x-axis actpos -------------------------------------------------------------- *)
	95	:	(* action:  *)
					IF	StepActionImPulse
						THEN
							AxisCtrl[AxisNo.XAxis].Command.OperationMode.CmdSetEncoderPosition		:=	TRUE;
							AxisCtrl[AxisNo.XAxis].Command.NominalValue.PositionSetNewEncoderPos	:=	0;
					END_IF;

					(* transition:  *)
					IF	StepAction AND
						(NOT StepActionImPulse) AND
						(NOT AxisCtrl[AxisNo.XAxis].Command.OperationMode.CmdSetEncoderPosition)
						THEN
							StepNew								:= 	100;							(* -> Activate safety state *)
					END_IF;
		(*------------------------------------------------------------Activate Safety state----------------------------------------------------------------*)
				(*Action*)

	100:			IF	StepActionImPulse
					THEN
						MachineCtrl.Peripheral.SafetyState.CmdActivate		:=	TRUE;
						MachineCtrl.ProcessControl.Event.En					:=	TRUE;
				END_IF;

				(*Transition*)
				IF	StepAction AND
				(NOT StepActionImPulse) AND
				( NOT MachineCtrl.Peripheral.SafetyState.CmdActivate ) AND
				MachineCtrl.state.SafetyState.unit.IsActive
					THEN
						StepNew	:= 110;								(* -> Message : Open Door*)
				END_IF;

		(* ------------------------------------------------ Message : Open Door&Set Up Mode---------------------------------------------------*)

				(*Action*)
	110:			IF	StepActionImPulse
					THEN
					(* set Event *)
						MachineCtrl.ProcessControl.Event.No			:=	EvNoOpenDoorInitSetUpMode;
						MachineCtrl.ProcessControl.Event.En			:=	TRUE;
						MachineCtrl.ProcessControl.Event.SId		:=	EvEventSourceId;
						MachineCtrl.ProcessControl.Event.Class		:=	TcEventClassMessage;
						MachineCtrl.Peripheral.Buzzer.Unit.CmdOn	:=	TRUE;
				END_IF;
				(* transition:  *)
				IF	StepAction AND
					(NOT StepActionImPulse) AND
					MachineCtrl.state.door.sharpener.IsOpen AND
					MachineCtrl.State.Mode.InitSetUp.IsActive
					THEN
						StepNew	:= 121;									(* desable Axis X&Z *)
				END_IF;

			(* ----------------------------------------------------------desable Axis-------------------------------------------------------------------- *)

	121:		(*Action*)
				IF	StepActionImPulse
					THEN
					(* set axis state for check *)
						AxisState	:=	STATE_DISABLED;
					(* Reset x-axis *)
						AxisCtrl[AxisNo.XAxis].Command.OperationMode.CmdPowerOn			:=	FALSE;
						AxisCtrl[AxisNo.XAxis].Command.OperationMode.CmdMoveAbsolut		:=	FALSE;
						AxisCtrl[AxisNo.XAxis].Command.OperationMode.CmdCamming			:=	FALSE;

					(* Reset Z-axis *)
						AxisCtrl[AxisNo.ZAxis].Command.OperationMode.CmdPowerOn			:=	FALSE;
						AxisCtrl[AxisNo.ZAxis].Command.OperationMode.CmdMoveAbsolut		:=	FALSE;
						AxisCtrl[AxisNo.ZAxis].Command.OperationMode.CmdCamming			:=	FALSE;
				END_IF;
				(*Transition*)
				(* status x-axis *)
				IF	StepAction AND
					(NOT StepActionImPulse) AND
					( Axis[AxisNo.XAxis].Status.Disabled)  AND
					(* status Z-axis *)
					( Axis[AxisNo.ZAxis].Status.Disabled)
					THEN
						StepNew		:=	123;								(*Deactivate Safety  while the door is open*)
				END_IF;

			(*------------------------------------------------Deactivate Safety  while the door is open--------------------------------------------*)

				(*Action*)
	123:			IF	StepActionImPulse
					THEN
						MachineCtrl.Peripheral.SafetyState.CmdDeactivate	:=	TRUE;
				END_IF;

				(*Wait for a While Before Activating Axis*)
				TONWaitSafetyStatePause( IN  	:=  	StepAction AND
												( NOT MachineCtrl.Peripheral.SafetyState.CmdDeactivate ) AND
												( NOT MachineCtrl.state.SafetyState.unit.IsActive ),
										 PT 	:= 	TIME#20ms);

				StartButton(CLK:= MachineCtrl.Peripheral.ExternalControl.StartSwitch , Q=> );

				(* transition:  *)
				IF	StepAction AND
					(NOT StepActionImPulse) AND
					MachineCtrl.state.SafetyState.unit.IsInactive AND
					(NOT MachineCtrl.Peripheral.SafetyState.CmdDeactivate) AND
					TONWaitSafetyStatePause.Q
					THEN
						StepNew		:=130;
				END_IF;
			(*--------------------------------------------------------------Activate Axis X-Z-------------------------------------------------------------*)

				(*Action*)
	130:			IF	StepActionImPulse
					THEN
						(* set axis state for check *)
						AxisState	:=	STATE_WAIT_NEWOPERATION;
						(*X-Axis*)
						AxisCtrl[AxisNo.XAxis].Command.OperationMode.CmdPowerOn					:=	TRUE;
						AxisCtrl[AxisNo.XAxis].Command.OperationMode.CmdJogHandwheel 				:=	FALSE;
						AxisCtrl[AxisNo.XAxis].Command.OperationMode.CmdJogButtonHandWheel		:=	FALSE;
						AxisCtrl[AxisNo.XAxis].Command.NominalValue.VeloJog						:=	ChipBreakerXAxisVelo;		(*XAxisVelo;*)
						AxisCtrl[AxisNo.XAxis].Command.ExternalControl.override						:=	100;

						(*Z-Axis*)

						AxisCtrl[AxisNo.ZAxis].Command.OperationMode.CmdPowerOn					:=	TRUE;
						AxisCtrl[AxisNo.ZAxis].Command.OperationMode.CmdJog						:=	FALSE;
						AxisCtrl[AxisNo.ZAxis].Command.OperationMode.CmdJogHandwheel				:=	FALSE;
						AxisCtrl[AxisNo.ZAxis].Command.NominalValue.VeloJog						:=	3;						(* 3 mm / second *)
						AxisCtrl[AxisNo.ZAxis].Command.ExternalControl.override						:=	100;
				END_IF;

				(*Transition*)
				IF	StepAction AND
					(NOT StepActionImPulse) AND
				(* operation mode *)
					MachineCtrl.State.Mode.InitSetUp.IsActive AND
				(* status x-axis *)
					(NOT Axis[AxisNo.XAxis].Status.Disabled) AND
					Axis[AxisNo.XAxis].Status.StandStill AND
					( AxisCtrl[AxisNo.XAxis].feedback.state.ActualFbState = AxisState ) AND
				(* status y-axis *)
					(NOT Axis[AxisNo.ZAxis].Status.Disabled) AND
					Axis[AxisNo.ZAxis].Status.StandStill AND
					( AxisCtrl[AxisNo.ZAxis].feedback.state.ActualFbState = AxisState )
					THEN
						StepNew		:=	135;		(* Move Z-Axis with Handwheel  & X-Axis with Side Buttons*)
					(*Buffer Actual Positions*)
						XPosition	:=	Axis[AxisNo.XAxis].NcToPlc.ActPos;
						ZPosition	:=	Axis[AxisNo.ZAxis].NcToPlc.ActPos;
				END_IF;

			(*-------------------------------------- Move Z-Axis with Handwheel  & X-Axis with Side Keys--------------------------------------------*)
				(*Action*)

	135:			IF	StepActionImPulse
						THEN
							(*----------------------------------------Velocity Calculation------------------------------------------------------*)
						(* calc sawblade circumference *)
							SBCircumference				:=	ActualSawBlade.Diameter*PI;
							(* max feedrate chip breaker  *)
							ChipBreakerAutoXAxisMaxVelo	:=	5.0;
						(* calc velo x-axis degree/s *)
							ChipBreakerAutoVeloTemp		:=	( 360.0 * ChipBreakerAutoXAxisMaxVelo ) / SBCircumference;
							ChipBreakerXAxisVelo			:=	ChipBreakerAutoVeloTemp	;
							(*---------------------------------------------------------------------------------------------------------------------------*)

							(* X-axis *)
							AxisCtrl[AxisNo.XAxis].Command.OperationMode.CmdJogHandwheel				:=	FALSE;
							AxisCtrl[AxisNo.XAxis].Command.OperationMode.CmdJogButtonHandWheel		:=	TRUE;
							AxisCtrl[AxisNo.XAxis].Command.NominalValue.VeloJog						:=	ChipBreakerXAxisVelo;
							(*Z-Axis*)
							AxisCtrl[AxisNo.ZAxis].Command.OperationMode.CmdJog						:=	FALSE;
							AxisCtrl[AxisNo.ZAxis].Command.OperationMode.CmdJogHandwheel				:=	TRUE;
							AxisCtrl[AxisNo.ZAxis].Command.NominalValue.VeloJog						:=	3;			(* 3 mm / second *)
							AxisCtrl[AxisNo.ZAxis].Command.ExternalControl.ExternalEncoderNumber			:=	AxisNo.ZAxisExtENC100.ExtEncNo;
							AxisCtrl[AxisNo.ZAxis].Command.ExternalControl.ExternalEncoderRatioNumerator	:=	18;
							AxisCtrl[AxisNo.ZAxis].Command.ExternalControl.ExternalEncoderRatioDenominator	:=	1;

							(*Moving X-Axis*)

							AxisCtrl[AxisNo.XAxis].Command.ExternalControl.StartPlus						:=	XMoveManual ;	(*With Side Keys*)

							(* status led touching *)
								MachineCtrl.Peripheral.ExternalControl.StatusLedOnTouch1	:=	TRUE;
								MachineCtrl.Peripheral.ExternalControl.StatusLedOnTouch2	:=	FALSE;

							(* set Event *)
								MachineCtrl.ProcessControl.Event.No		:=	EvNoProcessTouchingNo1;
								MachineCtrl.ProcessControl.Event.En		:=	TRUE;
								MachineCtrl.ProcessControl.Event.SId	:=	EvEventSourceId;
								MachineCtrl.ProcessControl.Event.Class	:=	TcEventClassMessage;
				END_IF;

				AxisCtrl[AxisNo.XAxis].Command.ExternalControl.StartPlus			:=	 MachineCtrl.Peripheral.ExternalControl.Key1Touching ;

			(*Transition*)
				IF	StepAction AND
					( NOT StepActionImPulse ) AND
					(* Confirm Touch Position  *)
					RTrigConfirmTouchposZ.Q
					THEN
						StepNew															:=	136;		(* action: Desable x + Z axis *)
				END_IF;

			(*--------------------------------------------------------------------- Clamping -----------------------------------------------------------------------*)
	136:			(*Action*)
				IF	StepActionImPulse
					THEN
						MachineCtrl.Peripheral.ChipBreaker.Auto.Clamping.CmdClose	:=	TRUE;
						MachineCtrl.Peripheral.ChipBreaker.Auto.Clamping.CmdOpen	:=	FALSE;
				END_IF;
				(*Transition*)
				IF	StepAction AND
					(NOT StepActionImPulse) AND
					MachineCtrl.State.ChipBreaker.Auto.Clamping.ClampingIsOn
					THEN
						StepNew			:=	138;
				END_IF;

				(*---------------------------------------Move The  Axis Manually while the SB is clamped-----------------------------------*)
	138:			(*Action*)
				IF	StepActionImPulse
						THEN
							(*----------------------------------------Velocity Calculation------------------------------------------------------*)
						(* calc sawblade circumference *)
							SBCircumference				:=	ActualSawBlade.Diameter*PI;
							(* max feedrate chip breaker  *)
							ChipBreakerAutoXAxisMaxVelo	:=	5.0;
						(* calc velo x-axis degree/s *)
							ChipBreakerAutoVeloTemp		:=	( 360.0 * ChipBreakerAutoXAxisMaxVelo ) / SBCircumference;
							ChipBreakerXAxisVelo			:=	ChipBreakerAutoVeloTemp	;
							(*---------------------------------------------------------------------------------------------------------------------------*)

							(* X-axis *)
							AxisCtrl[AxisNo.XAxis].Command.OperationMode.CmdJogHandwheel				:=	FALSE;
							AxisCtrl[AxisNo.XAxis].Command.OperationMode.CmdJogButtonHandWheel		:=	TRUE;
							AxisCtrl[AxisNo.XAxis].Command.NominalValue.VeloJog						:=	ChipBreakerXAxisVelo;
							(*Z-Axis*)
							AxisCtrl[AxisNo.ZAxis].Command.OperationMode.CmdJog						:=	FALSE;
							AxisCtrl[AxisNo.ZAxis].Command.OperationMode.CmdJogHandwheel				:=	TRUE;
							AxisCtrl[AxisNo.ZAxis].Command.NominalValue.VeloJog						:=	3;			(* 3 mm / second *)
							AxisCtrl[AxisNo.ZAxis].Command.ExternalControl.ExternalEncoderNumber			:=	AxisNo.ZAxisExtENC100.ExtEncNo;
							AxisCtrl[AxisNo.ZAxis].Command.ExternalControl.ExternalEncoderRatioNumerator	:=	36;
							AxisCtrl[AxisNo.ZAxis].Command.ExternalControl.ExternalEncoderRatioDenominator	:=	1;

							(*Moving X-Axis*)

							AxisCtrl[AxisNo.XAxis].Command.ExternalControl.StartPlus						:=	XMoveManual ;	(*With Side Keys*)

				END_IF;

				AxisCtrl[AxisNo.XAxis].Command.ExternalControl.StartPlus			:=	 MachineCtrl.Peripheral.ExternalControl.Key1Touching ;		(*Out Of Impulse so we can Move x Axis As long as not confirmed *)

				(*Transition*)

				IF	StepAction AND
					( NOT StepActionImPulse ) AND
					( NOT AxisCtrl[AxisNo.ZAxis].Command.OperationMode.CmdMoveAbsolut ) AND
					(NOT AxisCtrl[AxisNo.XAxis].Command.OperationMode.CmdMoveAbsolut) AND
					(* Confirm Touch Position  *)
					RTrigConfirmTouchposZ.Q
					THEN
						StepNew																		:=	140;		(* action: Desable x + Z axis *)
						(*Buuffer Z Position*)
						XPosition																	:=	Axis[AxisNo.XAxis].NcToPlc.ActPos;
						ZPosition																	:=	Axis[AxisNo.ZAxis].NcToPlc.ActPos;
						MachineCtrl.ProcessControl.Event.En												:=	FALSE;
						MachineCtrl.Peripheral.ExternalControl.StatusLedOnTouch1							:=	FALSE;
						MachineCtrl.Peripheral.ExternalControl.StatusLedOnTouch2							:=	FALSE;
						(* default Start X&Z-axis *)
						AxisCtrl[AxisNo.XAxis].Command.OperationMode.CmdJogHandwheel					:=	FALSE;
						AxisCtrl[AxisNo.XAxis].Command.OperationMode.CmdJogButtonHandWheel			:=	FALSE;
						AxisCtrl[AxisNo.ZAxis].Command.OperationMode.CmdJogHandwheel					:=	FALSE;
				END_IF;

			(*-------------------------------------------------------------------x-z axis Deactivation--------------------------------------------------------------*)

				(*Action*)
	140:			IF	StepActionImPulse
					THEN
					(* set axis state for check *)
						AxisState	:=	STATE_DISABLED;
						(*X-Axis*)
						AxisCtrl[AxisNo.XAxis].Command.OperationMode.CmdPowerOn						:=	FALSE;
						AxisCtrl[AxisNo.XAxis].Command.OperationMode.CmdMoveAbsolut					:=	FALSE;
						AxisCtrl[AxisNo.XAxis].Command.OperationMode.CmdJogButtonHandWheel			:=	FALSE;
						AxisCtrl[AxisNo.XAxis].Command.OperationMode.CmdJogHandwheel					:=	FALSE;
					(* Reset z-axis *)
						AxisCtrl[AxisNo.ZAxis].Command.OperationMode.CmdPowerOn						:=	FALSE;
						AxisCtrl[AxisNo.ZAxis].Command.OperationMode.CmdMoveAbsolut					:=	FALSE;
						AxisCtrl[AxisNo.ZAxis].Command.OperationMode.CmdJog							:=	FALSE;
						AxisCtrl[AxisNo.ZAxis].Command.OperationMode.CmdJogHandwheel					:=	FALSE;
				END_IF;

			(* transition *)

			IF	StepAction AND
				(NOT StepActionImPulse) AND
				(* all axis are disabled *)
					Axis[AxisNo.XAxis].Status.Disabled  AND
					Axis[AxisNo.ZAxis].Status.Disabled
				THEN
					StepNew	:= 150;				(* -> Activate Safety State*)
			END_IF;

		(* ---------------------------------------------------------------- Activate Safety State------------------------------------------------------------*)

			(*Action*)
	150:		IF	StepActionImPulse
				THEN
					MachineCtrl.Peripheral.SafetyState.CmdActivate	:=	TRUE;
			END_IF;

			(*Transition*)

			IF	StepAction AND
				(NOT StepActionImPulse)AND
				MachineCtrl.State.SafetyState.Unit.IsActive
				THEN
					StepNew		:=	160;	(*Event Close Door And Start*)
			END_IF;

			(*------------------------------------------------------Event Close Door And Start---------------------------------------------------------*)
			(*Action*)
	160:		IF	StepActionImPulse
				THEN
						MachineCtrl.ProcessControl.Event.No			:=	EvNoCloseDoorAutoMode;
						MachineCtrl.ProcessControl.Event.En			:=	TRUE;
						MachineCtrl.ProcessControl.Event.SId		:=	EvEventSourceId;
						MachineCtrl.ProcessControl.Event.Class		:=	TcEventClassMessage;
						MachineCtrl.Peripheral.Buzzer.Unit.CmdOn	:=	TRUE;
			END_IF;

			(*Transition*)

			IF	StepAction AND
				(NOT StepActionImPulse) AND
				MachineCtrl.State.Door.Sharpener.IsClosed AND
				MachineCtrl.State.Mode.Automatic.IsActive
				THEN
					StepNew		:=	165;		(*Deactivate safety state*)
					MachineCtrl.ProcessControl.Event.En		:=	FALSE;
			END_IF;
			(*-------------------------------------------Deactivate Safety State And Wait for Start Switch-------------------------------------*)
			(*Action*)
	165:		IF	StepActionImPulse
				THEN
						MachineCtrl.Peripheral.SafetyState.CmdDeactivate	:=	TRUE;
			END_IF;

				(*Wait for while after the Deactivation of  Safety state to avoid the error*)

				TONWaitSafetyStatePause( IN  	:=  	StepAction AND
												( NOT MachineCtrl.Peripheral.SafetyState.CmdDeactivate ) AND
												( NOT MachineCtrl.state.SafetyState.unit.IsActive ),
												 PT 	:= 	TIME#50ms);

				StartButton(CLK:= MachineCtrl.Peripheral.ExternalControl.StartSwitch , Q=> );

				(* transition:  *)
				IF	StepAction AND
					(NOT StepActionImPulse) AND
					NOT MachineCtrl.state.SafetyState.unit.IsActive  AND
					(NOT MachineCtrl.Peripheral.SafetyState.CmdDeactivate) AND
					TONWaitSafetyStatePause.Q
					THEN
						StepNew		:=170;
				END_IF;
			(*-----------------------------------------------------------Activation Of Axis X & Z---------------------------------------------------------------*)

				(*Action*)
  	 170:			IF	StepActionImPulse
					THEN
							(* set axis state for check *)
								AxisState	:=	STATE_WAIT_NEWOPERATION;
							(* x-axis - Enable *)
								AxisCtrl[AxisNo.XAxis].Command.OperationMode.CmdPowerOn			:=	TRUE;
								AxisCtrl[AxisNo.XAxis].Command.OperationMode.CmdMoveAbsolut		:=	FALSE;
								AxisCtrl[AxisNo.XAxis].Command.OperationMode.CmdCamming			:=	FALSE;
								AxisCtrl[AxisNo.XAxis].Command.ExternalControl.override				:=	100;
							(* Z-axis - Enable *)
								AxisCtrl[AxisNo.ZAxis].Command.OperationMode.CmdPowerOn			:=	TRUE;
								AxisCtrl[AxisNo.ZAxis].Command.OperationMode.CmdMoveAbsolut		:=	FALSE;
								AxisCtrl[AxisNo.ZAxis].Command.OperationMode.CmdCamming			:=	FALSE;
								AxisCtrl[AxisNo.ZAxis].Command.ExternalControl.override				:=	100;
				END_IF;

				(*Transition*)
				IF	StepAction AND
					(NOT StepActionImPulse) AND
					AutomaticMode AND
				(* status x-axis *)
					(NOT Axis[AxisNo.XAxis].Status.Disabled) AND
					Axis[AxisNo.XAxis].Status.StandStill AND
					( AxisCtrl[AxisNo.XAxis].feedback.state.ActualFbState = AxisState ) AND
				(* status Z-axis *)
					(NOT Axis[AxisNo.ZAxis].Status.Disabled) AND
					Axis[AxisNo.ZAxis].Status.StandStill AND
					( AxisCtrl[AxisNo.ZAxis].feedback.state.ActualFbState = AxisState ) AND
				(* stop switch not pressed *)
					(PauseSwitchActive)
					THEN
					StepNew	:= 	175;	(* --- move to   x-axis and Z-axis  To definiert positions------- *)
				END_IF;

				(*------------------------------------------------------Needed Calc For The Process--------------------------------------------------------*)
	175:			(*Action*)
				IF	StepActionImPulse
					THEN
							Zx						:=	UI.MachineSpecification.PeripheralOptional.ChipBreaker.ZPosCorrectionResharpRecut*2;
							(*degree per tooth calc*)
							DegPerTeeth			:=	(1/ UINT_TO_LREAL(UI.Order.SawBlade.NumberOfTeeth))  *360;
							(*UpfeedMM calc*)
							ZAxisUpfeedMM		:=
													2*(MachineCtrl.ProcessTemp.ActualJobData.Job.Infeed.TotalInfeed +
													REAL_TO_LREAL (UI.MachineSpecification.PeripheralOptional.ChipBreaker.YOffSet));
							RSS				:=	ActualGrindingWheel.Diameter / 2;
							DSSDiff				:=	200 - ActualGrindingWheel.Diameter;
							WorkingAngle		:=	UI.MachineSpecification.Base.WorkingAngle;
							BSS					:=	ActualGrindingWheel.Layer.Thickness;
							WorkingAngleRAD 	:=	WorkingAngle / 180 * PI;
							YrefPos				:=	YDistanceToTouchPos  -  UI.MachineSpecification.PeripheralBasic.Axis.Y.Position.HomingOffset;
							YendPos			:=	MachineCtrl.ProcessTemp.ActualJobData.OperatingMode.EndPosActOpMode.PosY;	;(* SFC Circular Grinding*)
							DeltaZ				:=	2*(YrefPos-YendPos)*COS(WorkingAngleRAD ) + Zx ;									(*Z-Axis Corrector : Zx*)
							DeltaX				:=	SIN(WorkingAngleRAD )*(YendPos - YrefPos -100+RSS) + 0.5*(BSS-2);
							DeltaX_DEG			:=	( 360.0 / (ActualSawBlade.Diameter * PI) ) * DeltaX;									(*DeltaX MM2DEG*)
							XoffsetInGrad			:=	( 360.0 / (ActualSawBlade.Diameter * PI) ) * UI.MachineSpecification.PeripheralOptional.ChipBreaker.XOffSet;
				END_IF;

				(*Transition*)
				IF	StepAction AND
					(NOT StepActionImPulse)
					THEN
						StepNew		:=	875;
				END_IF;
				(*#######################################END MANUELLE POS#############################################*)

				(*-------------------------------------------------------------Wait For User Interaction---------------------------------------------------*)
	875:			(*Action*)
				IF	StepActionImpulse
					THEN
						NextStepPulse	:=	TRUE;
				END_IF;

				IF	StepAction AND
					( RTrigNextStep.Q OR
					ContinousMode )
					THEN
						StepNew			:= 	880;
						NextStepPulse	:=	FALSE;
							IF	(   MachineCtrl.ProcessTemp.ActualJobData.SpecialTooth.TKCompensationActive)
								THEN
								XPosition		:=	Axis[AxisNo.XAxis].NcToPlc.ActPos;
							END_IF;
				END_IF;

				(* -------------------------------------- move to   x-axis and Z-axis  To defined  positions----------------------------------------- *)
	880	:		(* action  *)
					IF	StepActionImPulse
					THEN
							AxisState	:=	STATE_WAIT_NEWOPERATION;
						(* x-axis - move absolute *)
							AxisCtrl[AxisNo.XAxis].Command.OperationMode.CmdPowerOn			:=	TRUE;
							AxisCtrl[AxisNo.XAxis].Command.OperationMode.CmdJogHandwheel	 	:=	FALSE;
							AxisCtrl[AxisNo.XAxis].Command.OperationMode.CmdMoveAbsolut		:=	TRUE;
							AxisCtrl[AxisNo.XAxis].Command.OperationMode.CmdCamming			:=	FALSE;
							AxisCtrl[AxisNo.XAxis].Command.NominalValue.PositionMoveAbsolut		:=	XPosition;
							AxisCtrl[AxisNo.XAxis].Command.NominalValue.VeloMoveAbsolut		:=	3;							(* velocity To Definiert  x-axis Pos *)
							AxisCtrl[AxisNo.XAxis].Command.ExternalControl.override				:=	100;
						(* Z-axis - move absolute *)
							AxisCtrl[AxisNo.ZAxis].Command.OperationMode.CmdPowerOn			:=	TRUE;
							AxisCtrl[AxisNo.ZAxis].Command.OperationMode.CmdJogHandwheel 		:=	FALSE;
							AxisCtrl[AxisNo.ZAxis].Command.OperationMode.CmdMoveAbsolut		:=	TRUE;
							AxisCtrl[AxisNo.ZAxis].Command.OperationMode.CmdCamming			:=	FALSE;
							AxisCtrl[AxisNo.ZAxis].Command.NominalValue.PositionMoveAbsolut		:=	ZPosition;
							AxisCtrl[AxisNo.ZAxis].Command.NominalValue.VeloMoveAbsolut		:=	20;							(* velocity To Definiert  z-axis Pos *)
							AxisCtrl[AxisNo.ZAxis].Command.ExternalControl.override				:=	100;

							ActualRevolutions	:=	0;
					END_IF;

					(* transition:  *)
					IF	StepAction AND
						(NOT StepActionImPulse) AND
						(* status x-axis *)
							Axis[AxisNo.XAxis].Status.StandStill AND
							Axis[AxisNo.XAxis].Status.InTargetPosition AND
							( NOT AxisCtrl[AxisNo.XAxis].Command.OperationMode.CmdMoveAbsolut ) AND
							( AxisCtrl[AxisNo.XAxis].feedback.state.ActualFbState = AxisState ) AND
						(* status Z-axis *)
							Axis[AxisNo.ZAxis].Status.StandStill AND
							Axis[AxisNo.ZAxis].Status.InTargetPosition AND
							( NOT AxisCtrl[AxisNo.ZAxis].Command.OperationMode.CmdMoveAbsolut ) AND
							( AxisCtrl[AxisNo.ZAxis].feedback.state.ActualFbState = AxisState )
						THEN
							IF 	(NOT ManPosActive)
								THEN
									StepNew	:= 	883;			(* Close Clamping*)
								ELSE
									StepNew	:=	885;
							END_IF;
					END_IF;

			(* -------------------------------------- move to x-axis startpos ----------------------------------------- *)
			(* MachineCtrl.Peripheral.ChipBreaker.Auto.Number_Rev_Chamf.Rev_Chamfering *)
	883	:		(* action  *)
					IF	StepActionImPulse
					THEN
							AxisState	:=	STATE_WAIT_NEWOPERATION;
						(* x-axis - move absolute *)
							AxisCtrl[AxisNo.XAxis].Command.OperationMode.CmdPowerOn			:=	TRUE;
							AxisCtrl[AxisNo.XAxis].Command.OperationMode.CmdJogHandwheel	 	:=	FALSE;
							AxisCtrl[AxisNo.XAxis].Command.OperationMode.CmdMoveAbsolut		:=	TRUE;
							AxisCtrl[AxisNo.XAxis].Command.OperationMode.CmdCamming			:=	FALSE;

							IF	( NOT  MachineCtrl.ProcessTemp.ActualJobData.SpecialTooth.TKCompensationActive)
								THEN
									AxisCtrl[AxisNo.XAxis].Command.NominalValue.PositionMoveAbsolut		:=		AxisCtrl[AxisNo.XAxis].Command.NominalValue.PositionMoveAbsolut + DegPerTeeth - DeltaX_DEG + XoffsetInGrad;
									ELSE
										IF	(MachineCtrl.ProcessTemp.ActualJobData.OperatingMode.Previous= OperatingMode.Recutting) OR
											(MachineCtrl.ProcessTemp.ActualJobData.OperatingMode.Previous= OperatingMode.ReSharpening)
											THEN
												IF	 (MachineCtrl.ProcessTemp.ActualJobData.OperatingDirection.Previous = 'ClockWise')
													THEN
													(*cw previous*)
													AxisCtrl[AxisNo.XAxis].Command.NominalValue.PositionMoveAbsolut		:=      	Axis[AxisNo.XAxis].NcToPlc.ActPos  -
																															 AxisPhasingCAM.CbaTeethDiff[UI.Order.SawBlade.NumberOfTeeth] +
																															 DegPerTeeth -
																															DeltaX_DEG +
																															 XoffsetInGrad ;
													ELSE	(*ccw*)
													AxisCtrl[AxisNo.XAxis].Command.NominalValue.PositionMoveAbsolut		:=      	Axis[AxisNo.XAxis].NcToPlc.ActPos  -
																															 AxisPhasingCAM.CbaTeethDiff[UI.Order.SawBlade.NumberOfTeeth - 2] +
																															 DegPerTeeth -
																															DeltaX_DEG +
																															 XoffsetInGrad ;
												END_IF;
											ELSE
													;	 (* Hier Chamfering*)
												IF	(MachineCtrl.ProcessTemp.ActualJobData.OperatingMode.Previous= 'ChamferingAlternate') OR
													(MachineCtrl.ProcessTemp.ActualJobData.OperatingMode.Previous= 'ChamferingDual')
													THEN
														IF	 (MachineCtrl.ProcessTemp.ActualJobData.OperatingDirection.PreviousPrevious = 'ClockWise')
															THEN
																IF	 (MachineCtrl.ProcessTemp.ActualJobData.OperatingDirection.Previous  = 'ClockWise')
																	 THEN ;(*CW*)
																		AxisCtrl[AxisNo.XAxis].Command.NominalValue.PositionMoveAbsolut		:=      	MachineCtrl.ProcessTemp.ActualJobData.OperatingMode.EndPosActOpMode.PosX_CBA  -
																																				 AxisPhasingCAM.CbaTeethDiff[UI.Order.SawBlade.NumberOfTeeth] +
																																				 DegPerTeeth -
																																				DeltaX_DEG +
																																				 XoffsetInGrad -
																																				(360*2*MachineCtrl.Peripheral.ChipBreaker.Auto.Number_Rev_Chamf.Rev_Chamfering) ;
																		TestArray[0]	:= TRUE;
																	ELSE (*CCW*)
																		AxisCtrl[AxisNo.XAxis].Command.NominalValue.PositionMoveAbsolut		:=      	MachineCtrl.ProcessTemp.ActualJobData.OperatingMode.EndPosActOpMode.PosX_CBA  -
																																				 AxisPhasingCAM.CbaTeethDiff[UI.Order.SawBlade.NumberOfTeeth] +
																																				 DegPerTeeth -
																																				DeltaX_DEG +
																																				 XoffsetInGrad +
																																				(360*2*MachineCtrl.Peripheral.ChipBreaker.Auto.Number_Rev_Chamf.Rev_Chamfering) ;
																		TestArray[1]	:= TRUE;
																END_IF
															ELSE
																IF	 (MachineCtrl.ProcessTemp.ActualJobData.OperatingDirection.Previous  = 'ClockWise')
																	 THEN ;(*CW*)
																		AxisCtrl[AxisNo.XAxis].Command.NominalValue.PositionMoveAbsolut		:=      	MachineCtrl.ProcessTemp.ActualJobData.OperatingMode.EndPosActOpMode.PosX_CBA  -
																																				 AxisPhasingCAM.CbaTeethDiff[UI.Order.SawBlade.NumberOfTeeth - 2] +
																																				 DegPerTeeth -
																																				DeltaX_DEG +
																																				 XoffsetInGrad  -
																																				(360*2*MachineCtrl.Peripheral.ChipBreaker.Auto.Number_Rev_Chamf.Rev_Chamfering) ; ;
																		TestArray[2]	:= TRUE;
																	ELSE
																		AxisCtrl[AxisNo.XAxis].Command.NominalValue.PositionMoveAbsolut		:=      	MachineCtrl.ProcessTemp.ActualJobData.OperatingMode.EndPosActOpMode.PosX_CBA  -
																																				 AxisPhasingCAM.CbaTeethDiff[UI.Order.SawBlade.NumberOfTeeth - 2] +
																																				 DegPerTeeth -
																																				DeltaX_DEG +
																																				 XoffsetInGrad  +
																																				(360*2*MachineCtrl.Peripheral.ChipBreaker.Auto.Number_Rev_Chamf.Rev_Chamfering) ; ;
																		TestArray[3]	:= TRUE;
																END_IF;
														END_IF
												END_IF;
														(* Hier Chamfering*)
										END_IF;
	
								END_IF;

							AxisCtrl[AxisNo.XAxis].Command.NominalValue.VeloMoveAbsolut		:=	3;							(* velocity To Definiert  x-axis Pos *)
							AxisCtrl[AxisNo.XAxis].Command.ExternalControl.override				:=	100;
					END_IF;

					(* transition:  *)
					IF	StepAction AND
						(NOT StepActionImPulse) AND
						(* status x-axis *)
							Axis[AxisNo.XAxis].Status.StandStill AND
							Axis[AxisNo.XAxis].Status.InTargetPosition AND
							( NOT AxisCtrl[AxisNo.XAxis].Command.OperationMode.CmdMoveAbsolut ) AND
							( AxisCtrl[AxisNo.XAxis].feedback.state.ActualFbState = AxisState )
						THEN
							StepNew	:= 	885;			(* Close Clamping*)
					END_IF;

				(*---------------------------------------------------------Wait For User Interaction------------------------------------------------*)
	885:			IF	StepActionImpulse
					THEN
						NextStepPulse	:=	TRUE;
				END_IF;

				IF	StepAction AND
					( RTrigNextStep.Q OR
					ContinousMode )
					THEN
						StepNew			:= 	890;
						NextStepPulse	:=	FALSE;
						LimitZaxis		:=	Axis[AxisNo.ZAxis].NcToPlc.ActPos - 14;
				END_IF;

				(*-------------------------------------------------------Close- Clamping-----------------------------------------------------------------*)
	890:			(*Action*)
					IF	StepActionImPulse
						THEN
							MachineCtrl.Peripheral.ChipBreaker.Auto.Clamping.CmdClose	:=	TRUE;
							MachineCtrl.Peripheral.ChipBreaker.Auto.Clamping.CmdOpen	:=	FALSE;
					END_IF;

					TonWaitClamping(		IN	 :=	 StepAction AND
											MachineCtrl.State.ChipBreaker.Auto.Clamping.ClampingIsOn	,
											 PT	:= TIME#500ms,	(*2s*)
											Q=> , ET=> );

					(* transition:  *)
					IF	StepAction AND
						(NOT StepActionImPulse) AND
						(* clamping is open *)
						MachineCtrl.State.ChipBreaker.Auto.Clamping.ClampingIsOn AND
						TonWaitClamping.Q
						THEN
							StepNew	:= 	895;		(*Activation Of Turbine*)
					END_IF;

				(*--------------------------------------------------------Wait For User Interaction--------------------------------------------------------*)
	895:			IF	StepActionImpulse
					THEN
						NextStepPulse	:=	TRUE;
				END_IF;

				IF	StepAction AND
					( RTrigNextStep.Q OR
					ContinousMode )
					THEN
						StepNew			:= 	900;
						NextStepPulse	:=	FALSE;
				END_IF;

				(*----------------------------------------------------------- Turbine Activation-----------------------------------------------------------*)
	900:			(*Action : Activate Turbine#8*)

					IF	 StepActionImPulse
						THEN
								MachineCtrl.Peripheral.ChipBreaker.Auto.Turbine.CmdOn	:=	TRUE;
								MachineCtrl.Peripheral.ChipBreaker.Auto.Turbine.CmdOff	:=	FALSE;
								NumberTouch			:=	0;
								TriesNumber				:=	0;
					END_IF;

					(*Transition: Is the  Turbine On? *)

					IF	 StepAction 	AND
						 (NOT StepActionImPulse) AND
					    	  MachineCtrl.State.ChipBreaker.Auto.Turbine.IsActive AND
						  MachineCtrl.State.ChipBreaker.Auto.GrindingWheelIsReady
						THEN
							IF	Stepper  AND
								(NOT CbaPneumatic)
								THEN
									StepNew			:=	950	;		(*Servo- Motor *)
								ELSIF	CbaPneumatic AND
										(NOT Stepper)
										THEN
											StepNew		:=	990;		(*Pneumatic Cylinder *)
							END_IF;
							(*DemoMode ?*)
							IF  	UI.MachineSpecification.Base.DemoMode
								THEN
									StepNew				:=	1275;
									ZAxisStartPosition		:=	ZPosition - 4;
							END_IF;
					END_IF;


		(*-----------------------------------------Transition Servo Front/Rear Pos  #10 --------------------------------------------------*)
	950:			(*Action*)
					IF 	ChipBreakerFr
							THEN
								StepNew		:=	980;			(*ChipBreakerFront With Servo *)
								ELSIF	ChipBreakerRe
									THEN
										StepNew		:=	970;	(*ChipBreaker Rear  With Servo *)
					END_IF;
					(*Demo Mode No Need To Move The Stepper*)
					IF	UI.MachineSpecification.Base.DemoMode
						THEN
							StepNew		:=	1110;
					END_IF;
		(*#############################Chip Breaker Rear With Servo##############################-*)


  		(*------------------------------------------------------Wait For User Interaction----------------------------------------------------------*)
	970:			IF	StepActionImpulse
					THEN
						NextStepPulse	:=	TRUE;
				END_IF;

				IF	StepAction AND
					( RTrigNextStep.Q OR
					ContinousMode )
					THEN
						StepNew				:= 	 975;;
						NextStepPulse		:=	FALSE;
						StartMonitoringAaxis	:=	TRUE;
						StepMotorDestination	:=	ARearPos;
						AaxisActPosition		:=	 MachineCtrl.State.ChipBreaker.Auto.AaxisActualPos;
				END_IF;
		(*---------------------------------------------------Wait For Confirmation-----------------------------------------------------------*)
	9700:

				IF	RTrigNextStep.Q OR
					TRUE
					THEN
						StepNew	:= 9750;
				END_IF;

		(*-----------Move the A-Axis with a high velocity till it reaches the 80% of destination-----------------------*)

	9750:
				(*Action*)
				IF 	StepActionImpulse
					THEN
					AxisCtrl[AxisNo.AAxis].Command.OperationMode.CmdJog				:=	TRUE;
					AxisCtrl[AxisNo.AAxis].Command.ExternalControl.Override				:=	100;
					AxisCtrl[AxisNo.AAxis].Command.NominalValue.VeloJog				:=	0.2;
					AxisCtrl[AxisNo.AAxis].Command.ExternalControl.StartPlus				:=	FALSE;
					AxisCtrl[AxisNo.AAxis].Command.ExternalControl.StartMinus				:=	TRUE;
				END_IF;
				(*Transition*)
				IF 	StepAction AND
					(NOT StepActionImpulse) AND
					(MachineCtrl.State.ChipBreaker.Auto.AaxisActualPos <=  (ARear80 +AaxisTolerenceSlow)) AND
					(MachineCtrl.State.ChipBreaker.Auto.AaxisActualPos >=  (ARear80 -AaxisTolerenceSlow))
					THEN
						StepNew		:=	975;
						AxisCtrl[AxisNo.AAxis].Command.ExternalControl.StartMinus	:=	FALSE;
				END_IF;



	(*--------------------------------------------------------------Move X Axis One tooth----------------------------------------------------------*)

	1110:		(*Action*)
				IF	StepActionImpulse
					THEN
						AxisState														:=	STATE_WAIT_NEWOPERATION;
						AxisCtrl[AxisNo.XAxis].Command.OperationMode.CmdPowerOn			:=	TRUE;
						AxisCtrl[AxisNo.XAxis].Command.OperationMode.CmdMoveAbsolut		:=	TRUE;
						AxisCtrl[AxisNo.XAxis].Command.ExternalControl.override				:=	100;
						AxisCtrl[AxisNo.XAxis].Command.NominalValue.VeloMoveAbsolut		:=	3;
						AxisCtrl[AxisNo.XAxis].Command.OperationMode.CmdCamming			:=	FALSE;

						(*New*)
						MachineCtrl.Peripheral.ChipBreaker.Auto.Cooling.CmdOff				:=	FALSE;
						MachineCtrl.Peripheral.ChipBreaker.Auto.Cooling.CmdOn				:=	TRUE;



						IF	MachineCtrl.ProcessTemp.ActualJobData.SpecialTooth.VarioTooth.IsActive
							THEN																									(* first tooth pitch *)
								AxisCtrl[AxisNo.XAxis].Command.NominalValue.PositionMoveAbsolut		:=					Axis[AxisNo.XAxis].NcToPlc.ActPos +
																													FC_MM2DEG( 	MachineCtrl.ProcessTemp.ActualOrderStackBuffer.ActualOrder.SawBlade.Diameter,
																													MachineCtrl.ProcessTemp.ActualOrderStackBuffer.ActualOrder.SawBlade.Shape.ToothShape[0].ToothPitch.Absolute ) +
																													MachineCtrl.ProcessTemp.ActualJobData.SpecialTooth.VarioTooth.Distances.Front[VarioCtrEnd];
							ELSE
								(* Compensatoin not Active*)
								IF	(NOT MachineCtrl.ProcessTemp.ActualJobData.SpecialTooth.TKCompensationActive)
									THEN
										AxisCtrl[AxisNo.XAxis].Command.NominalValue.PositionMoveAbsolut				:= 	Axis[AxisNo.XAxis].NcToPlc.ActPos +
																													( 1 * DegPerTeeth );
										ELSE
										(*Test*)

										IF	(MachineCtrl.ProcessTemp.ActualJobData.OperatingMode.Previous= OperatingMode.Recutting) OR
											(MachineCtrl.ProcessTemp.ActualJobData.OperatingMode.Previous= OperatingMode.ReSharpening) OR
											(UI.Order.Job[1].OperatingMode =  OperatingMode.ReSharpening ) OR
											(UI.Order.Job[1].OperatingMode =  OperatingMode.Recutting )
											THEN
												IF	 (MachineCtrl.ProcessTemp.ActualJobData.OperatingDirection.Previous = 'ClockWise')
												  	  THEN
														   NoOfActTeethCompensation	:=	1 ; (*cw*)
													   ELSE
														   NoOfActTeethCompensation	:=	TO_INT(UI.Order.SawBlade.NumberOfTeeth) - 1;	(*ccw*)
												END_IF;
											ELSE
												(*Hier Chamfering*) ;
										END_IF;

										AxisCtrl[AxisNo.XAxis].Command.NominalValue.PositionMoveAbsolut				:=
																													Axis[AxisNo.XAxis].NcToPlc.ActPos +
																													( 1 * DegPerTeeth ) -
																													 AxisPhasingCAM.CbaTeethDiff[NoOfActTeethCompensation]	;



										XAxisNextPosition															:=	Axis[AxisNo.XAxis].NcToPlc.ActPos +
																													( 1 * DegPerTeeth ) -
																													 AxisPhasingCAM.CbaTeethDiff[NoOfActTeethCompensation]	;


								END_IF;
						END_IF;

				END_IF;
				(*Transition*)
				IF	StepAction AND
					NOT StepActionImPulse  AND
					(* status x-axis *)
					( NOT Axis[AxisNo.XAxis].Status.Disabled ) AND
					Axis[AxisNo.XAxis].Status.InTargetPosition AND
					( NOT AxisCtrl[AxisNo.XAxis].Command.OperationMode.CmdMoveAbsolut ) AND
					( AxisCtrl[AxisNo.XAxis].feedback.state.ActualFbState = AxisState )
					THEN
						StepNew		:=	1115;

						(* zero is the first element *)
						VarioCtr			:=	-1;
				END_IF;

	(*-----------------------------------------------------------------Keep Cooling On -------------------------------------------------------------------*)

	1115:		(*Action*)
				IF	StepActionImPulse
					THEN
						MachineCtrl.Peripheral.ChipBreaker.Auto.Cooling.CmdOff	:=	FALSE;(*TRUE;*)
						MachineCtrl.Peripheral.ChipBreaker.Auto.Cooling.CmdOn	:=	TRUE;

							IF	(MachineCtrl.ProcessTemp.ActualJobData.OperatingMode.Previous= OperatingMode.Recutting) OR
								(MachineCtrl.ProcessTemp.ActualJobData.OperatingMode.Previous= OperatingMode.ReSharpening) OR
								(UI.Order.Job[1].OperatingMode =  OperatingMode.ReSharpening ) OR
								(UI.Order.Job[1].OperatingMode =  OperatingMode.Recutting )
								THEN
									IF	 (MachineCtrl.ProcessTemp.ActualJobData.OperatingDirection.Previous = 'ClockWise')
										THEN
											NoOfActTeethCompensation	:=	TO_INT(UI.Order.SawBlade.NumberOfTeeth) ; (*cw*)
										ELSE
											NoOfActTeethCompensation	:=	TO_INT(UI.Order.SawBlade.NumberOfTeeth) - 2;  (*ccw*)
									END_IF;
							END_IF;
				END_IF;
				(*Transition*)
				IF	StepAction AND
					(NOT StepActionImPulse) AND
					MachineCtrl.State.ChipBreaker.Auto.Cooling.IsActive
					THEN
						StepNew		:=	1117;
				END_IF;
	(*---------------------------------------------------------------Wait For User Interaction-----------------------------------------------------------*)
	1117:		(*Action*)
				IF	StepActionImpulse
					THEN
						NextStepPulse	:=	TRUE;
				END_IF;
				(*Transition*)
				IF	StepAction AND
					( RTrigNextStep.Q OR
					ContinousMode )
					THEN
						StepNew			:= 	1120;
						NextStepPulse	:=	FALSE;
				END_IF;
	(*---------------------------------------------------------Transition Move Rear Position--------------------------------------------------------*)

	1120	:
				TON_Rear	(	 IN	:=	(StepNew = 1120) AND
										StepAction AND
										(NOT StepActionImPulse) AND
										ChipBreakerRe AND
										(NOT ChipBreakerFr),
										 PT	:=	T#1s ,
										 Q	=> ,
										 ET	=>						 );		(*---Wait 2 seconds before starting with the Rear Side-- *)

				(*Transition*)
				IF	StepAction AND
					(NOT StepActionImPulse) AND
					TON_Rear.Q
					THEN
						IF	Stepper AND
							(NOT CbaPneumatic )
							THEN
								MachineCtrl.Peripheral.ChipBreaker.Auto.TurbinePosition.CmdBackward	:=	FALSE;
								StepNew		:=	1290;
							ELSIF	 CbaPneumatic AND
									(NOT Stepper)
							THEN
								IF	NOT UI.MachineSpecification.Base.DemoMode
									THEN
										StepNew		:=	1125;
									ELSE
										StepNew		:=	1290;
								END_IF;
						END_IF;
				END_IF;
	(*---------------------------------------------------------------REAR-CYLINDRE-10--------------------------------------------------------------------*)
	1125	:		(*Action*)
					IF 	StepActionImpulse  AND
						(NOT MachineCtrl.State.ChipBreaker.Auto.TurbinePosition.InRearPosition) AND
						CbaPneumatic
					THEN
						MachineCtrl.Peripheral.ChipBreaker.Auto.TurbinePosition.CmdBackward	:=	TRUE;
						MachineCtrl.Peripheral.ChipBreaker.Auto.TurbinePosition.CmdForward	:=	FALSE;
					END_IF;

					(*Transition*)
					IF 	StepAction AND
						(NOT StepActionImpulse) AND
						(NOT MachineCtrl.Peripheral.ChipBreaker.Auto.TurbinePosition.CmdBackward) AND
						 MachineCtrl.State.ChipBreaker.Auto.TurbinePosition.InRearPosition
						THEN
							ZAxisStartPosition		:=	ZAxisStartPosition - UI.MachineSpecification.PeripheralOptional.ChipBreaker.ZDeltaFrontRearPos; (*0.05;*)
							XAxisEndPos			:=	Axis[AxisNo.XAxis].NcToPlc.ActPos  + 360;		(*Calc X Axis End Position*)
							StepNew				:=	1290;
					END_IF;

	(*---------------------------------------------------------------Wait For User Interaction-------------------------------------------------------*)
	1150:		(*Action*)
				IF	StepActionImpulse
					THEN
						NextStepPulse	:=	TRUE;
				END_IF;
				(*Transition*)
				IF	StepAction AND
					( RTrigNextStep.Q OR
					ContinousMode )
					THEN
						StepNew			:= 	1220;
						NextStepPulse	:=	FALSE;
				END_IF;
	(*----------------------------------------------------------Wait For User Interaction-------------------------------------------------------------*)
	1210:
				(*Action*)
				IF	StepActionImpulse
					THEN
						NextStepPulse	:=	TRUE;
				END_IF;
				(*Transition*)
				IF	StepAction AND
					( RTrigNextStep.Q OR
					ContinousMode )
					THEN
						StepNew			:= 	1215;
						NextStepPulse	:=	FALSE;
				END_IF;

	(*-----------------------If Double Touch Is Active and Number Of Touch <2:Z-Axis Move Down 3 MM-----------------------*)
	1215:
				(*Action*)
				IF 	StepActionImPulse
					THEN
						AxisState																:=	STATE_WAIT_NEWOPERATION;
						AxisCtrl[AxisNo.ZAxis].Command.OperationMode.CmdMoveAbsolut				:=	TRUE;
						AxisCtrl[AxisNo.ZAxis].Command.ExternalControl.override						:=	100;
						AxisCtrl[AxisNo.ZAxis].Command.OperationMode.CmdMoveAbsolutTouchProbe	:=	FALSE;		(*Down without Touch Probe :to not affect the touchnumber  *)
						AxisCtrl[AxisNo.ZAxis].Command.NominalValue.PositionMoveAbsolut				:= 	 Axis[AxisNo.ZAxis].NcToPlc.ActPos +3;
						AxisCtrl[AxisNo.ZAxis].Command.NominalValue.VeloMoveAbsolut				:=	1;
				END_IF;
				(*Transition*)
				IF	StepAction AND
					NOT StepActionImPulse  AND
					(* status z-axis *)
					( NOT Axis[AxisNo.ZAxis].Status.Disabled ) AND
					Axis[AxisNo.ZAxis].Status.InTargetPosition AND
					( NOT AxisCtrl[AxisNo.ZAxis].Command.OperationMode.CmdMoveAbsolut )AND
					( AxisCtrl[AxisNo.ZAxis].feedback.state.ActualFbState = AxisState )
					THEN
						StepNew		:=	1217;		(*User Interaction*)
				END_IF;
	(*------------------------------------------------------------Wait For User Interaction-------------------------------------------------------------------*)
	1217:		(*Action*)
				IF	StepActionImpulse
					THEN
						NextStepPulse	:=	TRUE;
				END_IF;
				(*Transition*)
				IF	StepAction AND
					( RTrigNextStep.Q OR
					ContinousMode )
					THEN
						StepNew			:= 	1220;
						NextStepPulse	:=	FALSE;
				END_IF;

	(*-------------------------------------------------------------------#11-- Z-Axis Move Up -----4 mm----------------------------------------------------*)
	1220	:		(*ACTION*)
					IF	StepActionImPulse
						THEN
							DifferenceMaxMinCBAGWDiameter												:=	 0.5 *
																											( UI.MachineSpecification.PeripheralOptional.ChipBreaker.GrindingWheel.Diameter.Maximal   -
																											 UI.MachineSpecification.PeripheralOptional.ChipBreaker.GrindingWheel.Diameter.Nominal );
							IF	(NOT UI.MachineSpecification.Base.DemoMode)
								THEN
									MachineCtrl.Peripheral.ChipBreaker.Auto.DustFan.CmdOn							:=	TRUE;
							END_IF;
							AxisCtrl[AxisNo.ZAxis].Command.OperationMode.CmdMoveAbsolutTouchProbe		:=	TRUE;
							AxisCtrl[AxisNo.ZAxis].Command.NominalValue.PositionMoveAbsolut					:= 	Axis[AxisNo.ZAxis].NcToPlc.ActPos -  14 (*7 is the org value*) - DifferenceMaxMinCBAGWDiameter;
	
							IF	(NumberTouch=0)
								THEN
									AxisCtrl[AxisNo.ZAxis].Command.NominalValue.VeloMoveAbsolut			:=	1;											 (*Velocity to Set*)
									ELSIF	(NumberTouch=1)
										THEN
											AxisCtrl[AxisNo.ZAxis].Command.NominalValue.VeloMoveAbsolut	:=	2;
							END_IF;
					END_IF;
					(*Transition: Did Z-Axis Reach The Grinding Wheel?*)
					IF 	StepAction AND
						(NOT StepActionImPulse) AND
						(NOT AxisCtrl[AxisNo.ZAxis].Command.OperationMode.CmdMoveAbsolutTouchProbe )

								THEN
									IF	( AxisCtrl[AxisNo.ZAxis].Feedback.State.TouchProbe.ActiveAndAxisStopped)
										THEN
												NumberTouch		:=	NumberTouch + 1;
											(*Calculation Of Number Of Touch*)
												IF	SimpleTouch
													THEN
														XAxisStartPosition													:=	Axis[AxisNo.XAxis].NcToPlc.ActPos;
														XAxisEndPos														:=	Axis[AxisNo.XAxis].NcToPlc.ActPos  + 360;		(*Calc X Axis End Position*)
														ZTouchPos														:=	Axis[AxisNo.ZAxis].NcToPlc.ActPos;
														ZAxisStartPosition													:=	ZTouchPos	+	0.7;							(*Move Z-Axis Down 0.7MM*)
														TouchPositionsZPlausi	[NumberTouch]								:=	Axis[AxisNo.ZAxis].NcToPlc.ActPos;				(*Touch Position Numbre*)
														AxisCtrl[AxisNo.ZAxis].Command.OperationMode.CmdMoveAbsolut		:=	FALSE;										(*End Moving Up of Z-Axis*)
														StepNew															:=	1245;										(*Z-Axis Down --> Start Pos*)
												END_IF;
												IF	DoubleTouch
												THEN
														IF	(NumberTouch<2)
															THEN
																StepNew		:=	1210;	(*Move Z Axis Down*)
																	ELSE	(*Touch >=2*)
																		ZTouchPos														:=	Axis[AxisNo.ZAxis].NcToPlc.ActPos;
																		ZAxisStartPosition													:=	ZTouchPos	+	0.7;
																		XAxisStartPosition													:=	Axis[AxisNo.XAxis].NcToPlc.ActPos;
																		XAxisEndPos														:=	Axis[AxisNo.XAxis].NcToPlc.ActPos  + 360;
																		AxisCtrl[AxisNo.ZAxis].Command.OperationMode.CmdMoveAbsolut		:=	FALSE;										(*End Moving Up of Z-Axis*)
																		StepNew															:=	1245;										(*Z-Axis Down --> Start Pos*)
														END_IF;
												END_IF;

								ELSE
											StepNew		:=	25000;;						(*If There is No Touch --> ERROR*)
											MachineCtrl.ProcessControl.Warning.No		:=	PSM_Fault_ErrorChipBreakerAuto;
											MachineCtrl.ProcessControl.Warning.En		:=	TRUE;
											MachineCtrl.Peripheral.Buzzer.Unit.CmdOn	:=	TRUE;
											MachineCtrl.ProcessControl.Warning.Data		:=	'';
					END_IF;
				END_IF;


	(*------------------------------------------------------------Wait For User Interaction-----------------------------------------------------*)

	1245:		(*Action*)
				IF	StepActionImpulse
					THEN
						NextStepPulse	:=	TRUE;
				END_IF;
				(*Transiiton*)
				IF	StepAction AND
					( RTrigNextStep.Q OR
					ContinousMode )
					THEN
						StepNew			:= 	1250;
						NextStepPulse	:=	FALSE;
				END_IF;
	(*---------------------------------------------------------------- Z-Axis Move Down---------------------------------------------------------*)

	1250:		(*Action*)
				IF 	StepActionImPulse
					THEN
						AxisCtrl[AxisNo.ZAxis].Command.OperationMode.CmdMoveAbsolut				:=	TRUE;;
						AxisCtrl[AxisNo.ZAxis].Command.NominalValue.PositionMoveAbsolut				:= 	ZAxisStartPosition  ;		  (*Moving down to start Pos*)
						AxisCtrl[AxisNo.ZAxis].Command.NominalValue.VeloMoveAbsolut				:=	10;
				END_IF;
				(*Transition :Is The Z-Axis in The  Position *)
				IF 	StepAction AND
					(NOT StepActionImPulse) AND
					(NOT AxisCtrl[AxisNo.ZAxis].Command.OperationMode.CmdMoveAbsolut)
					THEN
						DoubleTouch	:=	FALSE;
						IF	DoubleTouch
							THEN
								IF	(NumberTouch <2)
									THEN
										StepNew			:=	1255;			(*Move X-Axis 2 Teeth CCW then--> 122 Again:Move-Z UP*)
									ELSE									(*Number Of Touchs >=2*)
										(*Check Plausibility*)
										StepNew			:=	1265;			(*If OK-->Move X- Axis And Z-Axis To Start Position*)
									END_IF;
							ELSE
								StepNew			:=	1275;
						END_IF;
				END_IF;
	(*------------------------------------------------------------Wait For User Interaction-----------------------------------------------------*)
	1255:		(*Action*)
				IF	StepActionImpulse
					THEN
						NextStepPulse	:=	TRUE;
				END_IF;
				(*Transition*)
				IF	StepAction AND
					( RTrigNextStep.Q OR
					ContinousMode )
					THEN
						StepNew			:= 	1150;
						NextStepPulse	:=	FALSE;
				END_IF;

	(*------------------------------------------------------------Wait For User Interaction------------------------------------------------------*)
	1265:		(*Action*)
				IF	StepActionImpulse
					THEN
						NextStepPulse	:=	TRUE;
				END_IF;
				(*Transition*)
				IF	StepAction AND
					( RTrigNextStep.Q OR
					ContinousMode )
					THEN
						StepNew			:= 	1270;
						NextStepPulse	:=	FALSE;
				END_IF;

	(*------------------------------------------------------------------Check Plausibility-------------------------------------------------------------*)
	1270:			(*Action*)
					IF	DoubleTouch
						THEN
							Delta 	:=	ABS	 (TouchPositionsZPlausi[2]	-TouchPositionsZPlausi [1]);					(*Check Of Plausibility*)
							IF	(Delta <= DeltaMax)
							THEN
								StepNew						:=	1275;										(*Start POsition X/Z*)
								TouchPositionsPlausibilityOK 	:= 	TRUE;
								TouchPositionsPlausibilityError	:=	FALSE;
							ELSE
								TouchPositionsPlausibilityOK 	:= 	FALSE;
								TouchPositionsPlausibilityError	:=	TRUE;
								StepNew						:=	25000;										(*ERROR OUT*)
							END_IF;
					END_IF;
	(*-------------------------------------------------------------Wait For User Interaction------------------------------------------------------------*)
	1275:
				(*Action*)
				IF	StepActionImpulse
					THEN
						NextStepPulse	:=	TRUE;
				END_IF;
				(*Transition*)
				IF	StepAction AND
					( RTrigNextStep.Q OR
					ContinousMode )
					THEN
						StepNew			:= 	1280;
						NextStepPulse	:=	FALSE;
				END_IF;
	(*----------------------------------------------X-Axis & Z-Axis Move To Start Position A--#17----------------------------------------------*)
	1280	:		(*Action*)
					IF	StepActionImPulse
						THEN
							AxisState	:=	STATE_WAIT_NEWOPERATION;
							MachineCtrl.Peripheral.ChipBreaker.Auto.LowSpeedMonitoring.IsDeactivated	:=	TRUE;
						(* x-axis - move absolute *)
							AxisCtrl[AxisNo.XAxis].Command.OperationMode.CmdMoveAbsolut		:=	TRUE;
							AxisCtrl[AxisNo.XAxis].Command.OperationMode.CmdCamming			:=	FALSE;
							IF	(NOT UI.MachineSpecification.Base.DemoMode)
								THEN
									AxisCtrl[AxisNo.XAxis].Command.NominalValue.PositionMoveAbsolut		:=	XAxisStartPosition;			(* Startposition x-axis *)
							END_IF;
							AxisCtrl[AxisNo.XAxis].Command.NominalValue.VeloMoveAbsolut		:=	10;								(* velocity Startpos x-axis *)
							AxisCtrl[AxisNo.XAxis].Command.ExternalControl.override				:=	100;
						(* Z-axis - move absolute *)
							AxisCtrl[AxisNo.ZAxis].Command.OperationMode.CmdPowerOn			:=	TRUE;
							AxisCtrl[AxisNo.ZAxis].Command.OperationMode.CmdJogHandwheel 		:=	FALSE;
							AxisCtrl[AxisNo.ZAxis].Command.OperationMode.CmdMoveAbsolut		:=	TRUE;
							AxisCtrl[AxisNo.ZAxis].Command.OperationMode.CmdCamming			:=	FALSE;
							AxisCtrl[AxisNo.ZAxis].Command.NominalValue.PositionMoveAbsolut		:=	ZAxisStartPosition;			(* Startposition y-axis *)
							AxisCtrl[AxisNo.ZAxis].Command.NominalValue.VeloMoveAbsolut		:=	10;						(* velocity Startpos z-axis *)
							AxisCtrl[AxisNo.ZAxis].Command.ExternalControl.override				:=	100;
							XAxisNextPosition													:=	AxisCtrl[AxisNo.XAxis].Command.NominalValue.PositionMoveAbsolut;

							IF	(MachineCtrl.ProcessTemp.ActualJobData.OperatingMode.Previous= OperatingMode.Recutting) OR
								(MachineCtrl.ProcessTemp.ActualJobData.OperatingMode.Previous= OperatingMode.ReSharpening) OR
								(UI.Order.Job[1].OperatingMode =  OperatingMode.ReSharpening ) OR
								(UI.Order.Job[1].OperatingMode =  OperatingMode.Recutting )
								THEN
									IF	 (MachineCtrl.ProcessTemp.ActualJobData.OperatingDirection.Previous = 'ClockWise')
										THEN
											NoOfActTeethCompensation	:=		TO_INT(UI.Order.SawBlade.NumberOfTeeth) -1 ;				(*previous cw*)
										ELSE
											NoOfActTeethCompensation	:=		TO_INT(UI.Order.SawBlade.NumberOfTeeth) - 3;				(* previous ccw	 *)
									END_IF;
								ELSE
									(*Hier Chamfering *) ;
							END_IF;

					END_IF;

					(*Transition : Is X /Z Axis in Start Position*)

					IF 	StepAction AND
						(NOT StepActionImPulse) AND
						(* status x-axis *)
							Axis[AxisNo.XAxis].Status.StandStill AND
							Axis[AxisNo.XAxis].Status.InTargetPosition AND
							( NOT AxisCtrl[AxisNo.XAxis].Command.OperationMode.CmdMoveAbsolut ) AND
							( AxisCtrl[AxisNo.XAxis].feedback.state.ActualFbState = AxisState ) AND
						(* status Z-axis *)
							Axis[AxisNo.ZAxis].Status.StandStill AND
							Axis[AxisNo.ZAxis].Status.InTargetPosition AND
							( NOT AxisCtrl[AxisNo.ZAxis].Command.OperationMode.CmdMoveAbsolut ) AND
							( AxisCtrl[AxisNo.ZAxis].feedback.state.ActualFbState = AxisState )
					THEN
						StepNew			:=	1290;	(*Z-Axis UpFeed*)
						StartWriting		:=	TRUE;
					END_IF;
	(*-------------------------------------------------------------Wait For User Interaction------------------------------------------------------*)
	1290:	(*Action*)
			IF	StepActionImPulse
				THEN
					IF	MachineCtrl.ProcessTemp.ActualJobData.SpecialTooth.VarioTooth.IsActive
						THEN
							FOR	VarioCtr := 0 TO 11
									DO
										VarioToothPitch[VarioCtr]	:=	FC_MM2DEG( 	MachineCtrl.ProcessTemp.ActualOrderStackBuffer.ActualOrder.SawBlade.Diameter,
																					MachineCtrl.ProcessTemp.ActualOrderStackBuffer.ActualOrder.SawBlade.Shape.ToothShape[VarioCtr].ToothPitch.Absolute );

							END_FOR;

							VarioCtrEnd	:=	( ( MachineCtrl.ProcessTemp.ActualJobData.SpecialTooth.VarioTooth.ToothNo ) / 2 ) - 1;

